// TIA Portal V20 export
FUNCTION_BLOCK "CallEquipment"   // FB131, LAD
TITLE = CallEquipment
// Template of an equipment module. This block contains the logic and futher calls (e.g. sequences, control modules, diagnostics etc.) of the equipment module.
// It can be used out of the box but also adapted to your own needs.
// stored: IsIECCheckEnabled true, MemoryReserve 100, Namespace Unit1.Em2, SetENOAutomatically true
   VAR_INPUT
      ZoneOperationEnable { ExternalWritable := 'False'} : "LWONIK_typeSafetyZoneManualOperation";
      unitEnableControlInterfaces { ExternalWritable := 'False'} : "LAF_typeEnableControlInterfaces";
      commandExcute { ExternalWritable := 'False'} : Bool;
   END_VAR
   VAR_IN_OUT
      unitStatus : "LAF_typeUnitStatus";   // Current unit status o be used in this EM
      emFeedback : "LUC_typeEmFeedback";   // Feedback of the EM to the Unit
      unitAlarmDB : "LAF_typeAlarms";   // Summarized EM Alarms for the Unit
   END_VAR
   VAR
      instSequenceSemiAutoSplice { ExternalWritable := 'False'} : "Unit1.Em2.Sequence_1_SemiAutoSplice";
      instTapeUnitInitializedJob1 { ExternalWritable := 'False'} : "LAF_SelectJob";
      instAutoSplicerModuleInitializedJob2 { ExternalWritable := 'False'} : "LAF_SelectJob";
      instLeftSplicingModuleMoverInitializedJob3 { ExternalWritable := 'False'} : "LAF_SelectJob";
      instRightSplicingModuleMoverInitializedJob4 { ExternalWritable := 'False'} : "LAF_SelectJob";
      instSplicingModuleMoverAutoJob5 { ExternalWritable := 'False'} : "LAF_SelectJob";
      instVacuumAutoJob7 { ExternalWritable := 'False'} : "LAF_SelectJob";
      instCutterAutoJob8 { ExternalWritable := 'False'} : "LAF_SelectJob";
      instLeftElectrodeReMoverAutoJob9 { ExternalWritable := 'False'} : "LAF_SelectJob";
      instRightElectrodeReMoverAutoJob10 { ExternalWritable := 'False'} : "LAF_SelectJob";
      instTapeAttachReadyAutoJob11 { ExternalWritable := 'False'} : "LAF_SelectJob";
      instTapeAttachStartAutoJob12 { ExternalWritable := 'False'} : "LAF_SelectJob";
      instTapeAttachFinishAutoJob13 { ExternalWritable := 'False'} : "LAF_SelectJob";
      instLeftSplicingModuleMoverAutoJob14 { ExternalWritable := 'False'} : "LAF_SelectJob";
      instRightSplicingModuleMoverAutoJob15 { ExternalWritable := 'False'} : "LAF_SelectJob";
      instSemiAutoSpliceFullAutoJob20 { ExternalWritable := 'False'} : "LAF_SelectJob";
      instElectrodeFixRightTopFwdBwd { ExternalWritable := 'False'} : "LBC_TwoWayActuatorCn";
      instElectrodeFixRightBottomFwdBwd { ExternalWritable := 'False'} : "LBC_TwoWayActuatorCn";
      instElectrodeFixLeftTopFwdBwd { ExternalWritable := 'False'} : "LBC_TwoWayActuatorCn";
      instElectrodeFixLeftBottomFwdBwd { ExternalWritable := 'False'} : "LBC_TwoWayActuatorCn";
      instElectrodeFixLeftTopUpDown { ExternalWritable := 'False'} : "LBC_TwoWayActuatorCn";
      instElectrodeFixLeftBottomUpDown { ExternalWritable := 'False'} : "LBC_TwoWayActuatorCn";
      instUwSemiSplicerVacuumRightTopOnOff { ExternalWritable := 'False'} : "LBC_TwoWayActuatorCn";
      instUwSemiSplicerVacuumRightBottomOnOff { ExternalWritable := 'False'} : "LBC_TwoWayActuatorCn";
      instUwSemiSplicerVacuumLeftTopOnOff { ExternalWritable := 'False'} : "LBC_TwoWayActuatorCn";
      instUwSemiSplicerVacuumLeftBottomOnOff { ExternalWritable := 'False'} : "LBC_TwoWayActuatorCn";
      instElectrodeCutterFwdBwd { ExternalWritable := 'False'} : "LBC_TwoWayActuatorCn";
      instSplicingLeftModuleMoverFwdBwd { ExternalWritable := 'False'} : "LBC_TwoWayActuatorCn";
      instSplicingRightModuleMoverFwdBwd { ExternalWritable := 'False'} : "LBC_TwoWayActuatorCn";
      instElectrodeLeftHolderMoverFwdBwd { ExternalWritable := 'False'} : "LBC_TwoWayActuatorCn";
      instElectrodeRightHolderMoverFwdBwd { ExternalWritable := 'False'} : "LBC_TwoWayActuatorCn";
      instTapeLoadingTurnCwCcw { ExternalWritable := 'False'} : "LBC_TwoWayActuatorCn";
      instTapeAttachUnitFwdBwd { ExternalWritable := 'False'} : "LBC_TwoWayActuatorCn";
      instTapeVacuumOnOff { ExternalWritable := 'False'} : "LBC_TwoWayActuatorCn";
      instStopperFwdBwd { ExternalWritable := 'False'} : "LBC_TwoWayActuatorCn";
      instSupportUnitTransferFwdBwd { ExternalWritable := 'False'} : "LBC_TwoWayActuatorCn";
      instSupportUnitShaftUpDown { ExternalWritable := 'False'} : "LBC_TwoWayActuatorCn";
      instFrameCoverFwdBwd { ExternalWritable := 'False'} : "LBC_TwoWayActuatorCn";
      statUnitStatus { ExternalWritable := 'False'} : "LAF_typeUnitStatus";   // Unit Status used in this EM
      instManageAlarms { ExternalWritable := 'False'} : "LAF_ManageAlarms";
      instEventsPFE { S7_SetPoint := 'True'} : "Unit1.Em2.EventsPFE";
      JobSummary { ExternalWritable := 'False'} : "LAF_typeJobStatus";
      statEnableManualCmds { ExternalWritable := 'False'} : Bool;
      statPulse { ExternalWritable := 'False'} : Array[0..99] of Bool;
      statTonTimer { ExternalWritable := 'False'} : Array[0..99] of TON_TIME;
      statTofTimer { ExternalWritable := 'False'} : Array[0..99] of TOF_TIME;
      citi_Ptrig : Array[0..20] of Bool;
      citiTon : Array[0..20] of TON_TIME;
      citi : Time;
      citiTest : Array[0..20] of Bool;
   END_VAR
   VAR_TEMP
      tempScInProduction : Bool;   // Mode Production and StateComplete
      tempScNoProduction : Bool;   // Mode Manual and StateComplete
   END_VAR
   VAR CONSTANT
      TO_DO_INSERT_PRECONDITIONS_HERE : Bool := TRUE;   // Template : Add em specific conditions here
      NO_JOB : DInt;   // No job
      TRUE : Bool := TRUE;
      FALSE : Bool := FALSE;
   END_VAR
   VAR_TEMP   // added for the SCL form of the ladder/FBD networks
      _w1 : Bool;
      _w2 : Bool;
   END_VAR
BEGIN

REGION Network 1: BLOCK INFO HEADER
   // (company) / (C) Copyright (year)
   // ---------------------------------------------------------------------------------
   // Title:                             (Title of this block)
   // Comment/Function: (that is implemented in the block)
   // Library/Family:           (that the source is dedicated to)
   // Author:                        (department / person in charge / contact)
   // Target System:          (test system with FW version)
   // Engineering:              TIA Portal (SW version)
   // Restrictions:               (OB types, etc.)
   // Requirements:           (hardware, technological package, etc.)
   // ---------------------------------------------------------------------------------
   // Change log table:
   // Version          | Date             | Signature      | Expert in charge  | Changes applied ------------------------|----------------------|-------------------------|--------------------------------|-----------------------
   // 001.000.000 | yyyy-mm-dd | 0x00000000 | (name of expert) | First released version
END_REGION

REGION Network 2: DESCRIPTION
   // This is a template block provided by the Automation Framework. It can be used to create an own project.
   // The Block Info Header is prepared to put in your own data.
   // Description of the block could be added here and the docu created by Code2Docu.
END_REGION

REGION Network 3: ******************** Equipment Control ********************
END_REGION

REGION Network 4: Interlink EM to Unit
   // This block links and unlinks the EM from the unit. The command to link/unlink can be set directly by the inputs of the block (e.g. to link/unlink based on any program logic) or through the InOut "hmiInterface". The block changes the output "isLinked" to true/false, depending on the command and if a change is allowed. A changed is allowed if the unit is in state aborted, clearing or stopped. The output "isLinked" is send back to the unit. If the EM is not linked, the unit ignores this EM.
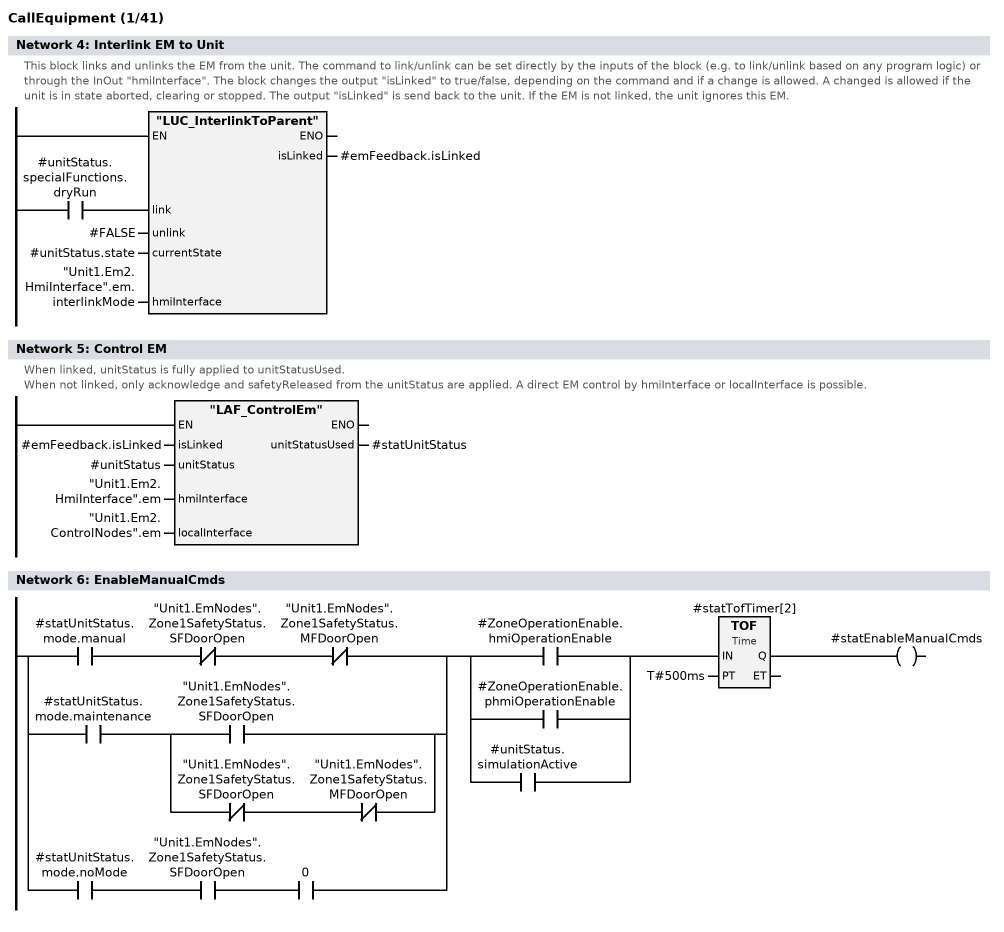
   RUNG wire#powerrail
      "LUC_InterlinkToParent"(link := wire#w1, unlink := #FALSE, currentState := #unitStatus.state, hmiInterface := "Unit1.Em2.HmiInterface".em.interlinkMode, isLinked => #emFeedback.isLinked)
   END_RUNG
   RUNG wire#powerrail
      Contact( #unitStatus.specialFunctions.dryRun )
   END_RUNG wire#w1
   // the same network as SCL:
   "LUC_InterlinkToParent"(link := #unitStatus.specialFunctions.dryRun,
                           unlink := #FALSE,
                           currentState := #unitStatus.state,
                           hmiInterface := "Unit1.Em2.HmiInterface".em.interlinkMode,
                           isLinked => #emFeedback.isLinked);
END_REGION

REGION Network 5: Control EM
   // When linked, unitStatus is fully applied to unitStatusUsed.
   // When not linked, only acknowledge and safetyReleased from the unitStatus are applied. A direct EM control by hmiInterface or localInterface is possible.
   RUNG wire#powerrail
      "LAF_ControlEm"(isLinked := #emFeedback.isLinked, unitStatus := #unitStatus, hmiInterface := "Unit1.Em2.HmiInterface".em, localInterface := "Unit1.Em2.ControlNodes".em, unitStatusUsed => #statUnitStatus)
   END_RUNG
   // the same network as SCL:
   "LAF_ControlEm"(isLinked := #emFeedback.isLinked,
                   unitStatus := #unitStatus,
                   hmiInterface := "Unit1.Em2.HmiInterface".em,
                   localInterface := "Unit1.Em2.ControlNodes".em,
                   unitStatusUsed => #statUnitStatus);
END_REGION

REGION Network 6: EnableManualCmds
   RUNG wire#powerrail
      Contact( #statUnitStatus.mode.manual )
      I_Contact( "Unit1.EmNodes".Zone1SafetyStatus.SFDoorOpen )
      I_Contact( "Unit1.EmNodes".Zone1SafetyStatus.MFDoorOpen )
      wire#w1
      Contact( #ZoneOperationEnable.hmiOperationEnable )
      wire#w3
      { S7_Templates := "time_type := Time" } #statTofTimer[2].TOF(pt := T#500ms, et =>)
      Coil( #statEnableManualCmds )
   END_RUNG
   RUNG wire#powerrail
      Contact( #statUnitStatus.mode.maintenance )
      wire#w2
      Contact( "Unit1.EmNodes".Zone1SafetyStatus.SFDoorOpen )
   END_RUNG wire#w1
   RUNG wire#w2
      I_Contact( "Unit1.EmNodes".Zone1SafetyStatus.SFDoorOpen )
      I_Contact( "Unit1.EmNodes".Zone1SafetyStatus.MFDoorOpen )
   END_RUNG wire#w1
   RUNG wire#powerrail
      Contact( #statUnitStatus.mode.noMode )
      Contact( "Unit1.EmNodes".Zone1SafetyStatus.SFDoorOpen )
      Contact( 0 )
   END_RUNG wire#w1
   RUNG wire#w1
      Contact( #ZoneOperationEnable.phmiOperationEnable )
   END_RUNG wire#w3
   RUNG wire#w1
      Contact( #unitStatus.simulationActive )
   END_RUNG wire#w3
   // the same network as SCL:
   #statTofTimer[2].TOF(IN := ((#statUnitStatus.mode.manual AND NOT "Unit1.EmNodes".Zone1SafetyStatus.SFDoorOpen AND NOT "Unit1.EmNodes".Zone1SafetyStatus.MFDoorOpen) OR (#statUnitStatus.mode.maintenance AND ("Unit1.EmNodes".Zone1SafetyStatus.SFDoorOpen OR (NOT "Unit1.EmNodes".Zone1SafetyStatus.SFDoorOpen AND NOT "Unit1.EmNodes".Zone1SafetyStatus.MFDoorOpen))) OR (#statUnitStatus.mode.noMode AND "Unit1.EmNodes".Zone1SafetyStatus.SFDoorOpen AND 0)) AND (#ZoneOperationEnable.hmiOperationEnable OR #ZoneOperationEnable.phmiOperationEnable OR #unitStatus.simulationActive),
                        PT := T#500ms);
   #statEnableManualCmds := #statTofTimer[2].Q;
END_REGION

REGION Network 7: Alarms Disabled
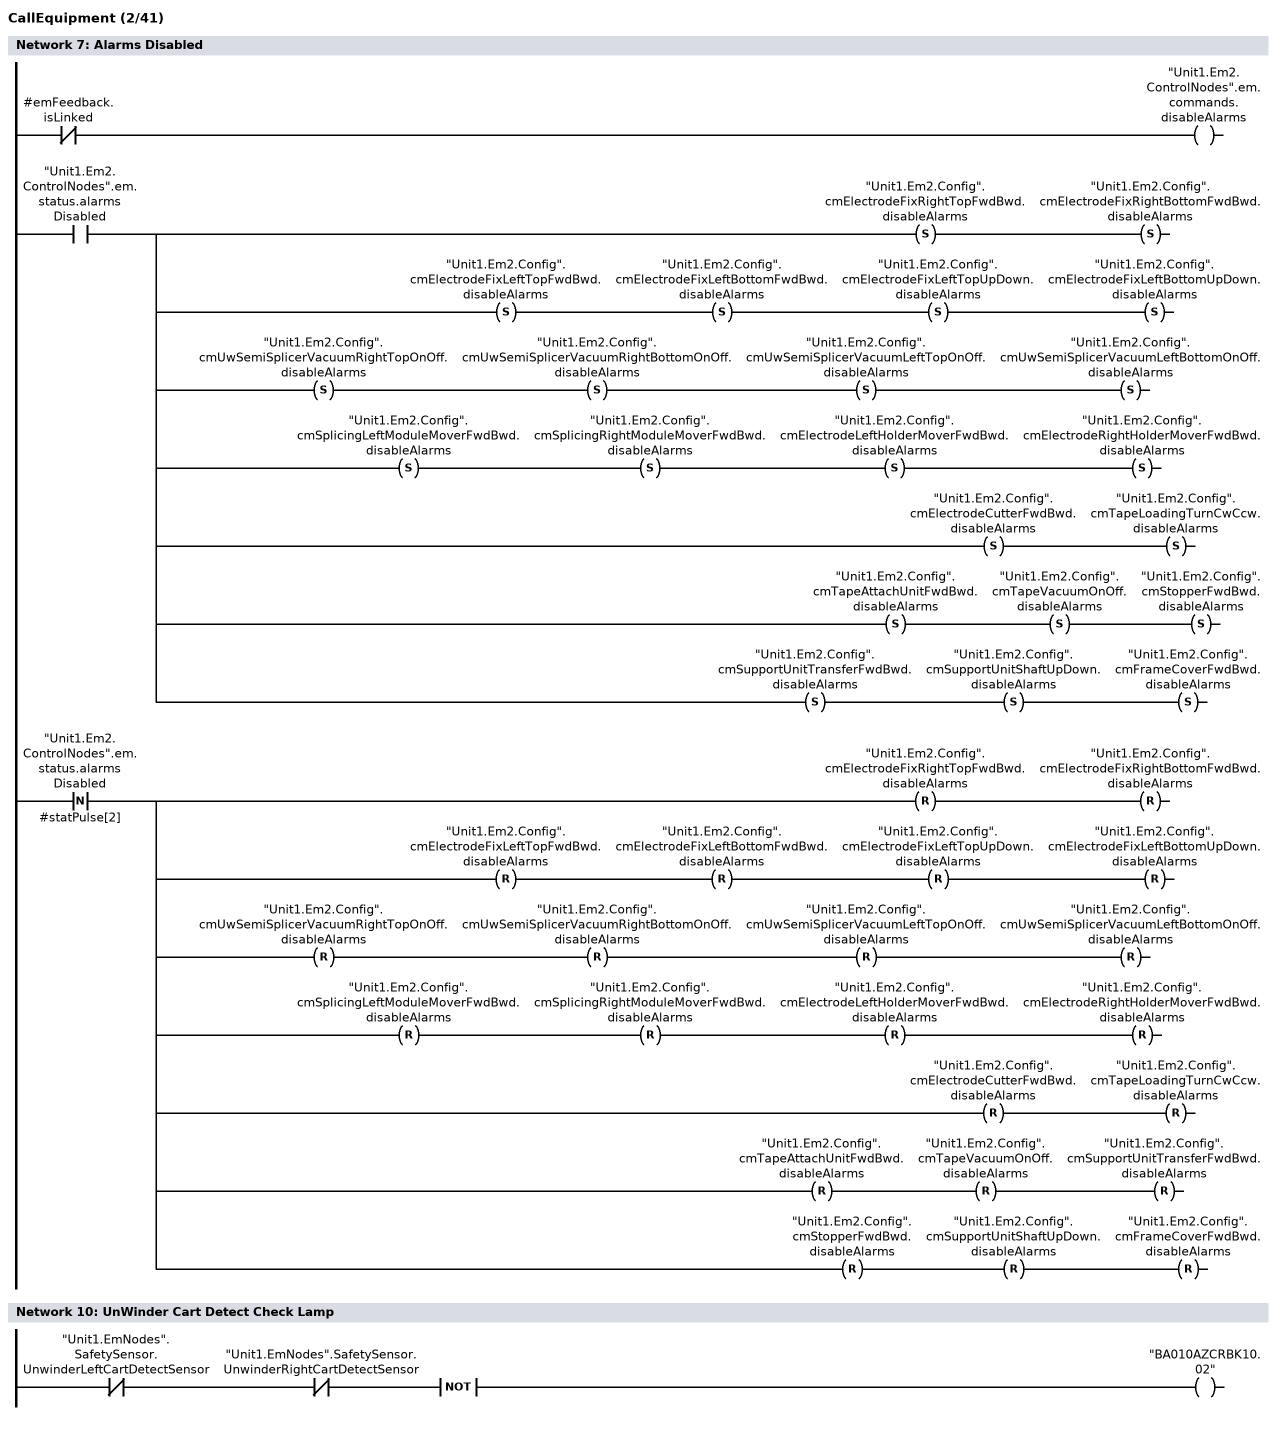
   RUNG wire#powerrail
      I_Contact( #emFeedback.isLinked )
      Coil( "Unit1.Em2.ControlNodes".em.commands.disableAlarms )
   END_RUNG
   RUNG wire#powerrail
      Contact( "Unit1.Em2.ControlNodes".em.status.alarmsDisabled )
      wire#w1
      S_Coil( "Unit1.Em2.Config".cmElectrodeFixRightTopFwdBwd.disableAlarms )
      S_Coil( "Unit1.Em2.Config".cmElectrodeFixRightBottomFwdBwd.disableAlarms )
   END_RUNG
   RUNG wire#w1
      S_Coil( "Unit1.Em2.Config".cmElectrodeFixLeftTopFwdBwd.disableAlarms )
      S_Coil( "Unit1.Em2.Config".cmElectrodeFixLeftBottomFwdBwd.disableAlarms )
      S_Coil( "Unit1.Em2.Config".cmElectrodeFixLeftTopUpDown.disableAlarms )
      S_Coil( "Unit1.Em2.Config".cmElectrodeFixLeftBottomUpDown.disableAlarms )
   END_RUNG
   RUNG wire#w1
      S_Coil( "Unit1.Em2.Config".cmUwSemiSplicerVacuumRightTopOnOff.disableAlarms )
      S_Coil( "Unit1.Em2.Config".cmUwSemiSplicerVacuumRightBottomOnOff.disableAlarms )
      S_Coil( "Unit1.Em2.Config".cmUwSemiSplicerVacuumLeftTopOnOff.disableAlarms )
      S_Coil( "Unit1.Em2.Config".cmUwSemiSplicerVacuumLeftBottomOnOff.disableAlarms )
   END_RUNG
   RUNG wire#w1
      S_Coil( "Unit1.Em2.Config".cmSplicingLeftModuleMoverFwdBwd.disableAlarms )
      S_Coil( "Unit1.Em2.Config".cmSplicingRightModuleMoverFwdBwd.disableAlarms )
      S_Coil( "Unit1.Em2.Config".cmElectrodeLeftHolderMoverFwdBwd.disableAlarms )
      S_Coil( "Unit1.Em2.Config".cmElectrodeRightHolderMoverFwdBwd.disableAlarms )
   END_RUNG
   RUNG wire#w1
      S_Coil( "Unit1.Em2.Config".cmElectrodeCutterFwdBwd.disableAlarms )
      S_Coil( "Unit1.Em2.Config".cmTapeLoadingTurnCwCcw.disableAlarms )
   END_RUNG
   RUNG wire#w1
      S_Coil( "Unit1.Em2.Config".cmTapeAttachUnitFwdBwd.disableAlarms )
      S_Coil( "Unit1.Em2.Config".cmTapeVacuumOnOff.disableAlarms )
      S_Coil( "Unit1.Em2.Config".cmStopperFwdBwd.disableAlarms )
   END_RUNG
   RUNG wire#w1
      S_Coil( "Unit1.Em2.Config".cmSupportUnitTransferFwdBwd.disableAlarms )
      S_Coil( "Unit1.Em2.Config".cmSupportUnitShaftUpDown.disableAlarms )
      S_Coil( "Unit1.Em2.Config".cmFrameCoverFwdBwd.disableAlarms )
   END_RUNG
   RUNG wire#powerrail
      N_Contact(operand := "Unit1.Em2.ControlNodes".em.status.alarmsDisabled, bit := #statPulse[2])
      wire#w2
      R_Coil( "Unit1.Em2.Config".cmElectrodeFixRightTopFwdBwd.disableAlarms )
      R_Coil( "Unit1.Em2.Config".cmElectrodeFixRightBottomFwdBwd.disableAlarms )
   END_RUNG
   RUNG wire#w2
      R_Coil( "Unit1.Em2.Config".cmElectrodeFixLeftTopFwdBwd.disableAlarms )
      R_Coil( "Unit1.Em2.Config".cmElectrodeFixLeftBottomFwdBwd.disableAlarms )
      R_Coil( "Unit1.Em2.Config".cmElectrodeFixLeftTopUpDown.disableAlarms )
      R_Coil( "Unit1.Em2.Config".cmElectrodeFixLeftBottomUpDown.disableAlarms )
   END_RUNG
   RUNG wire#w2
      R_Coil( "Unit1.Em2.Config".cmUwSemiSplicerVacuumRightTopOnOff.disableAlarms )
      R_Coil( "Unit1.Em2.Config".cmUwSemiSplicerVacuumRightBottomOnOff.disableAlarms )
      R_Coil( "Unit1.Em2.Config".cmUwSemiSplicerVacuumLeftTopOnOff.disableAlarms )
      R_Coil( "Unit1.Em2.Config".cmUwSemiSplicerVacuumLeftBottomOnOff.disableAlarms )
   END_RUNG
   RUNG wire#w2
      R_Coil( "Unit1.Em2.Config".cmSplicingLeftModuleMoverFwdBwd.disableAlarms )
      R_Coil( "Unit1.Em2.Config".cmSplicingRightModuleMoverFwdBwd.disableAlarms )
      R_Coil( "Unit1.Em2.Config".cmElectrodeLeftHolderMoverFwdBwd.disableAlarms )
      R_Coil( "Unit1.Em2.Config".cmElectrodeRightHolderMoverFwdBwd.disableAlarms )
   END_RUNG
   RUNG wire#w2
      R_Coil( "Unit1.Em2.Config".cmElectrodeCutterFwdBwd.disableAlarms )
      R_Coil( "Unit1.Em2.Config".cmTapeLoadingTurnCwCcw.disableAlarms )
   END_RUNG
   RUNG wire#w2
      R_Coil( "Unit1.Em2.Config".cmTapeAttachUnitFwdBwd.disableAlarms )
      R_Coil( "Unit1.Em2.Config".cmTapeVacuumOnOff.disableAlarms )
      R_Coil( "Unit1.Em2.Config".cmSupportUnitTransferFwdBwd.disableAlarms )
   END_RUNG
   RUNG wire#w2
      R_Coil( "Unit1.Em2.Config".cmStopperFwdBwd.disableAlarms )
      R_Coil( "Unit1.Em2.Config".cmSupportUnitShaftUpDown.disableAlarms )
      R_Coil( "Unit1.Em2.Config".cmFrameCoverFwdBwd.disableAlarms )
   END_RUNG
   // the same network as SCL:
   "Unit1.Em2.ControlNodes".em.commands.disableAlarms := NOT #emFeedback.isLinked;
   IF "Unit1.Em2.ControlNodes".em.status.alarmsDisabled THEN
       "Unit1.Em2.Config".cmElectrodeFixRightTopFwdBwd.disableAlarms := TRUE;
       "Unit1.Em2.Config".cmElectrodeFixRightBottomFwdBwd.disableAlarms := TRUE;
       "Unit1.Em2.Config".cmElectrodeFixLeftTopFwdBwd.disableAlarms := TRUE;
       "Unit1.Em2.Config".cmElectrodeFixLeftBottomFwdBwd.disableAlarms := TRUE;
       "Unit1.Em2.Config".cmElectrodeFixLeftTopUpDown.disableAlarms := TRUE;
       "Unit1.Em2.Config".cmElectrodeFixLeftBottomUpDown.disableAlarms := TRUE;
       "Unit1.Em2.Config".cmUwSemiSplicerVacuumRightTopOnOff.disableAlarms := TRUE;
       "Unit1.Em2.Config".cmUwSemiSplicerVacuumRightBottomOnOff.disableAlarms := TRUE;
       "Unit1.Em2.Config".cmUwSemiSplicerVacuumLeftTopOnOff.disableAlarms := TRUE;
       "Unit1.Em2.Config".cmUwSemiSplicerVacuumLeftBottomOnOff.disableAlarms := TRUE;
       "Unit1.Em2.Config".cmSplicingLeftModuleMoverFwdBwd.disableAlarms := TRUE;
       "Unit1.Em2.Config".cmSplicingRightModuleMoverFwdBwd.disableAlarms := TRUE;
       "Unit1.Em2.Config".cmElectrodeLeftHolderMoverFwdBwd.disableAlarms := TRUE;
       "Unit1.Em2.Config".cmElectrodeRightHolderMoverFwdBwd.disableAlarms := TRUE;
       "Unit1.Em2.Config".cmElectrodeCutterFwdBwd.disableAlarms := TRUE;
       "Unit1.Em2.Config".cmTapeLoadingTurnCwCcw.disableAlarms := TRUE;
       "Unit1.Em2.Config".cmTapeAttachUnitFwdBwd.disableAlarms := TRUE;
       "Unit1.Em2.Config".cmTapeVacuumOnOff.disableAlarms := TRUE;
       "Unit1.Em2.Config".cmStopperFwdBwd.disableAlarms := TRUE;
       "Unit1.Em2.Config".cmSupportUnitTransferFwdBwd.disableAlarms := TRUE;
       "Unit1.Em2.Config".cmSupportUnitShaftUpDown.disableAlarms := TRUE;
       "Unit1.Em2.Config".cmFrameCoverFwdBwd.disableAlarms := TRUE;
   END_IF;
   #_w1 := NOT "Unit1.Em2.ControlNodes".em.status.alarmsDisabled AND #statPulse[2];   // falling edge of "Unit1.Em2.ControlNodes".em.status.alarmsDisabled
   #statPulse[2] := "Unit1.Em2.ControlNodes".em.status.alarmsDisabled;
   IF #_w1 THEN
       "Unit1.Em2.Config".cmElectrodeFixRightTopFwdBwd.disableAlarms := FALSE;
       "Unit1.Em2.Config".cmElectrodeFixRightBottomFwdBwd.disableAlarms := FALSE;
       "Unit1.Em2.Config".cmElectrodeFixLeftTopFwdBwd.disableAlarms := FALSE;
       "Unit1.Em2.Config".cmElectrodeFixLeftBottomFwdBwd.disableAlarms := FALSE;
       "Unit1.Em2.Config".cmElectrodeFixLeftTopUpDown.disableAlarms := FALSE;
       "Unit1.Em2.Config".cmElectrodeFixLeftBottomUpDown.disableAlarms := FALSE;
       "Unit1.Em2.Config".cmUwSemiSplicerVacuumRightTopOnOff.disableAlarms := FALSE;
       "Unit1.Em2.Config".cmUwSemiSplicerVacuumRightBottomOnOff.disableAlarms := FALSE;
       "Unit1.Em2.Config".cmUwSemiSplicerVacuumLeftTopOnOff.disableAlarms := FALSE;
       "Unit1.Em2.Config".cmUwSemiSplicerVacuumLeftBottomOnOff.disableAlarms := FALSE;
       "Unit1.Em2.Config".cmSplicingLeftModuleMoverFwdBwd.disableAlarms := FALSE;
       "Unit1.Em2.Config".cmSplicingRightModuleMoverFwdBwd.disableAlarms := FALSE;
       "Unit1.Em2.Config".cmElectrodeLeftHolderMoverFwdBwd.disableAlarms := FALSE;
       "Unit1.Em2.Config".cmElectrodeRightHolderMoverFwdBwd.disableAlarms := FALSE;
       "Unit1.Em2.Config".cmElectrodeCutterFwdBwd.disableAlarms := FALSE;
       "Unit1.Em2.Config".cmTapeLoadingTurnCwCcw.disableAlarms := FALSE;
       "Unit1.Em2.Config".cmTapeAttachUnitFwdBwd.disableAlarms := FALSE;
       "Unit1.Em2.Config".cmTapeVacuumOnOff.disableAlarms := FALSE;
       "Unit1.Em2.Config".cmSupportUnitTransferFwdBwd.disableAlarms := FALSE;
       "Unit1.Em2.Config".cmStopperFwdBwd.disableAlarms := FALSE;
       "Unit1.Em2.Config".cmSupportUnitShaftUpDown.disableAlarms := FALSE;
       "Unit1.Em2.Config".cmFrameCoverFwdBwd.disableAlarms := FALSE;
   END_IF;
END_REGION

REGION Network 8 (SCL): ReferenceDesignator
   IF "Unit1.EmNodes".unitRecipe.processUnitNo = 2 THEN
       "Unit1.Em2.Config".cmElectrodeFixRightTopFwdBwd.referenceDesignator := WSTRING#'Electrode Fix Right Top';
       "Unit1.Em2.Config".cmElectrodeFixRightBottomFwdBwd.referenceDesignator := WSTRING#'Electrode Fix Right BTM';
       "Unit1.Em2.Config".cmElectrodeFixLeftTopFwdBwd.referenceDesignator := WSTRING#'Electrode Fix Left Top';
       "Unit1.Em2.Config".cmElectrodeFixLeftBottomFwdBwd.referenceDesignator := WSTRING#'Electrode Fix Left BTM';
       "Unit1.Em2.Config".cmElectrodeFixLeftTopUpDown.referenceDesignator := WSTRING#'Electrode Fix Left Top';
       "Unit1.Em2.Config".cmElectrodeFixLeftBottomUpDown.referenceDesignator := WSTRING#'Electrode Fix Left BTM';
       "Unit1.Em2.Config".cmUwSemiSplicerVacuumRightTopOnOff.referenceDesignator := WSTRING#'Splicer Vacuum Right Top';
       "Unit1.Em2.Config".cmUwSemiSplicerVacuumRightBottomOnOff.referenceDesignator := WSTRING#'Splicer Vacuum Right BTM';
       "Unit1.Em2.Config".cmUwSemiSplicerVacuumLeftTopOnOff.referenceDesignator := WSTRING#'Splicer Vacuum Left Top';
       "Unit1.Em2.Config".cmUwSemiSplicerVacuumLeftBottomOnOff.referenceDesignator := WSTRING#'Splicer Vacuum Left BTM';
       "Unit1.Em2.Config".cmElectrodeCutterFwdBwd.referenceDesignator := WSTRING#'Electrode Cutter';
       "Unit1.Em2.Config".cmSplicingLeftModuleMoverFwdBwd.referenceDesignator := WSTRING#'Left Module Mover';
       "Unit1.Em2.Config".cmSplicingRightModuleMoverFwdBwd.referenceDesignator := WSTRING#'Right Module Mover';
       "Unit1.Em2.Config".cmElectrodeLeftHolderMoverFwdBwd.referenceDesignator := WSTRING#'Left Holder Mover';
       "Unit1.Em2.Config".cmElectrodeRightHolderMoverFwdBwd.referenceDesignator := WSTRING#'Right Holder Mover';
       "Unit1.Em2.Config".cmTapeLoadingTurnCwCcw.referenceDesignator := WSTRING#'Tape Loading Tum';
       "Unit1.Em2.Config".cmTapeAttachUnitFwdBwd.referenceDesignator := WSTRING#'Tape Attach Unit';
       "Unit1.Em2.Config".cmTapeVacuumOnOff.referenceDesignator := WSTRING#'Tape Vacuum';
       "Unit1.Em2.Config".cmStopperFwdBwd.referenceDesignator := WSTRING#'Stopper';
       "Unit1.Em2.Config".cmSupportUnitTransferFwdBwd.referenceDesignator := WSTRING#'Support Unit Transfer';
       "Unit1.Em2.Config".cmSupportUnitShaftUpDown.referenceDesignator := WSTRING#'Support Unit Shaft';
       "Unit1.Em2.Config".cmFrameCoverFwdBwd.referenceDesignator := WSTRING#'Frame Cover';
   END_IF;

   IF "Unit1.EmNodes".unitRecipe.processUnitNo = 1 THEN
       "Unit1.Em2.Config".cmElectrodeFixRightTopFwdBwd.referenceDesignator := WSTRING#'Electrode Fix Left Top';
       "Unit1.Em2.Config".cmElectrodeFixRightBottomFwdBwd.referenceDesignator := WSTRING#'Electrode Fix Left BTM';
       "Unit1.Em2.Config".cmElectrodeFixLeftTopFwdBwd.referenceDesignator := WSTRING#'Electrode Fix Right Top';
       "Unit1.Em2.Config".cmElectrodeFixLeftBottomFwdBwd.referenceDesignator := WSTRING#'Electrode Fix Right BTM';
       "Unit1.Em2.Config".cmElectrodeFixLeftTopUpDown.referenceDesignator := WSTRING#'Electrode Fix Right Top';
       "Unit1.Em2.Config".cmElectrodeFixLeftBottomUpDown.referenceDesignator := WSTRING#'Electrode Fix Right BTM';
       "Unit1.Em2.Config".cmUwSemiSplicerVacuumRightTopOnOff.referenceDesignator := WSTRING#'Splicer Vacuum Left Top';
       "Unit1.Em2.Config".cmUwSemiSplicerVacuumRightBottomOnOff.referenceDesignator := WSTRING#'Splicer Vacuum Left BTM';
       "Unit1.Em2.Config".cmUwSemiSplicerVacuumLeftTopOnOff.referenceDesignator := WSTRING#'Splicer Vacuum Right Top';
       "Unit1.Em2.Config".cmUwSemiSplicerVacuumLeftBottomOnOff.referenceDesignator := WSTRING#'Splicer Vacuum Right BTM';
       "Unit1.Em2.Config".cmElectrodeCutterFwdBwd.referenceDesignator := WSTRING#'Electrode Cutter';
       "Unit1.Em2.Config".cmSplicingLeftModuleMoverFwdBwd.referenceDesignator := WSTRING#'Right Module Mover';
       "Unit1.Em2.Config".cmSplicingRightModuleMoverFwdBwd.referenceDesignator := WSTRING#'Left Module Mover';
       "Unit1.Em2.Config".cmElectrodeLeftHolderMoverFwdBwd.referenceDesignator := WSTRING#'Right Holder Mover';
       "Unit1.Em2.Config".cmElectrodeRightHolderMoverFwdBwd.referenceDesignator := WSTRING#'Left Holder Mover';
       "Unit1.Em2.Config".cmTapeLoadingTurnCwCcw.referenceDesignator := WSTRING#'Tape Loading Tum';
       "Unit1.Em2.Config".cmTapeAttachUnitFwdBwd.referenceDesignator := WSTRING#'Tape Attach Unit';
       "Unit1.Em2.Config".cmTapeVacuumOnOff.referenceDesignator := WSTRING#'Tape Vacuum';
       "Unit1.Em2.Config".cmStopperFwdBwd.referenceDesignator := WSTRING#'Stopper';
       "Unit1.Em2.Config".cmSupportUnitTransferFwdBwd.referenceDesignator := WSTRING#'Support Unit Transfer';
       "Unit1.Em2.Config".cmSupportUnitShaftUpDown.referenceDesignator := WSTRING#'Support Unit Shaft';
       "Unit1.Em2.Config".cmFrameCoverFwdBwd.referenceDesignator := WSTRING#'Frame Cover';
   END_IF;
END_REGION

REGION Network 9: ******************** Control Modules (Sensors) ********************
   // Call control modules that are sensors before the em logic (jobs and sequence), so that the latest value is used in the logic.
END_REGION

REGION Network 10: UnWinder Cart Detect Check Lamp
   RUNG wire#powerrail
      I_Contact( "Unit1.EmNodes".SafetySensor.UnwinderLeftCartDetectSensor )
      I_Contact( "Unit1.EmNodes".SafetySensor.UnwinderRightCartDetectSensor )
      Not()
      Coil( "BA010AZCRBK10.02" )
   END_RUNG
   // the same network as SCL:
   "BA010AZCRBK10.02" := NOT (NOT "Unit1.EmNodes".SafetySensor.UnwinderLeftCartDetectSensor AND NOT "Unit1.EmNodes".SafetySensor.UnwinderRightCartDetectSensor);
END_REGION

REGION Network 11: ******************** Equipment Logic ********************
   // Title:
   // Comment/Function:
   // Author:
   // Engineering:
   // Restrictions:
   // Requirements:
END_REGION

REGION Network 12: Map Unit Status to Sequence Status [1] Semi Auto Splice
   // This block maps the unit status to the seuqnce status. Thus, it controls the sequence depending on the unit status. E.g. it sets the sequence to automatic when the unit state is in productions. This blocks work perfectly with the sequences provided in the AF. 
   // This typed block (MapUnitStatusToSequence) could be adjusted to specific application requirements or if other, user-defined sequences are used.
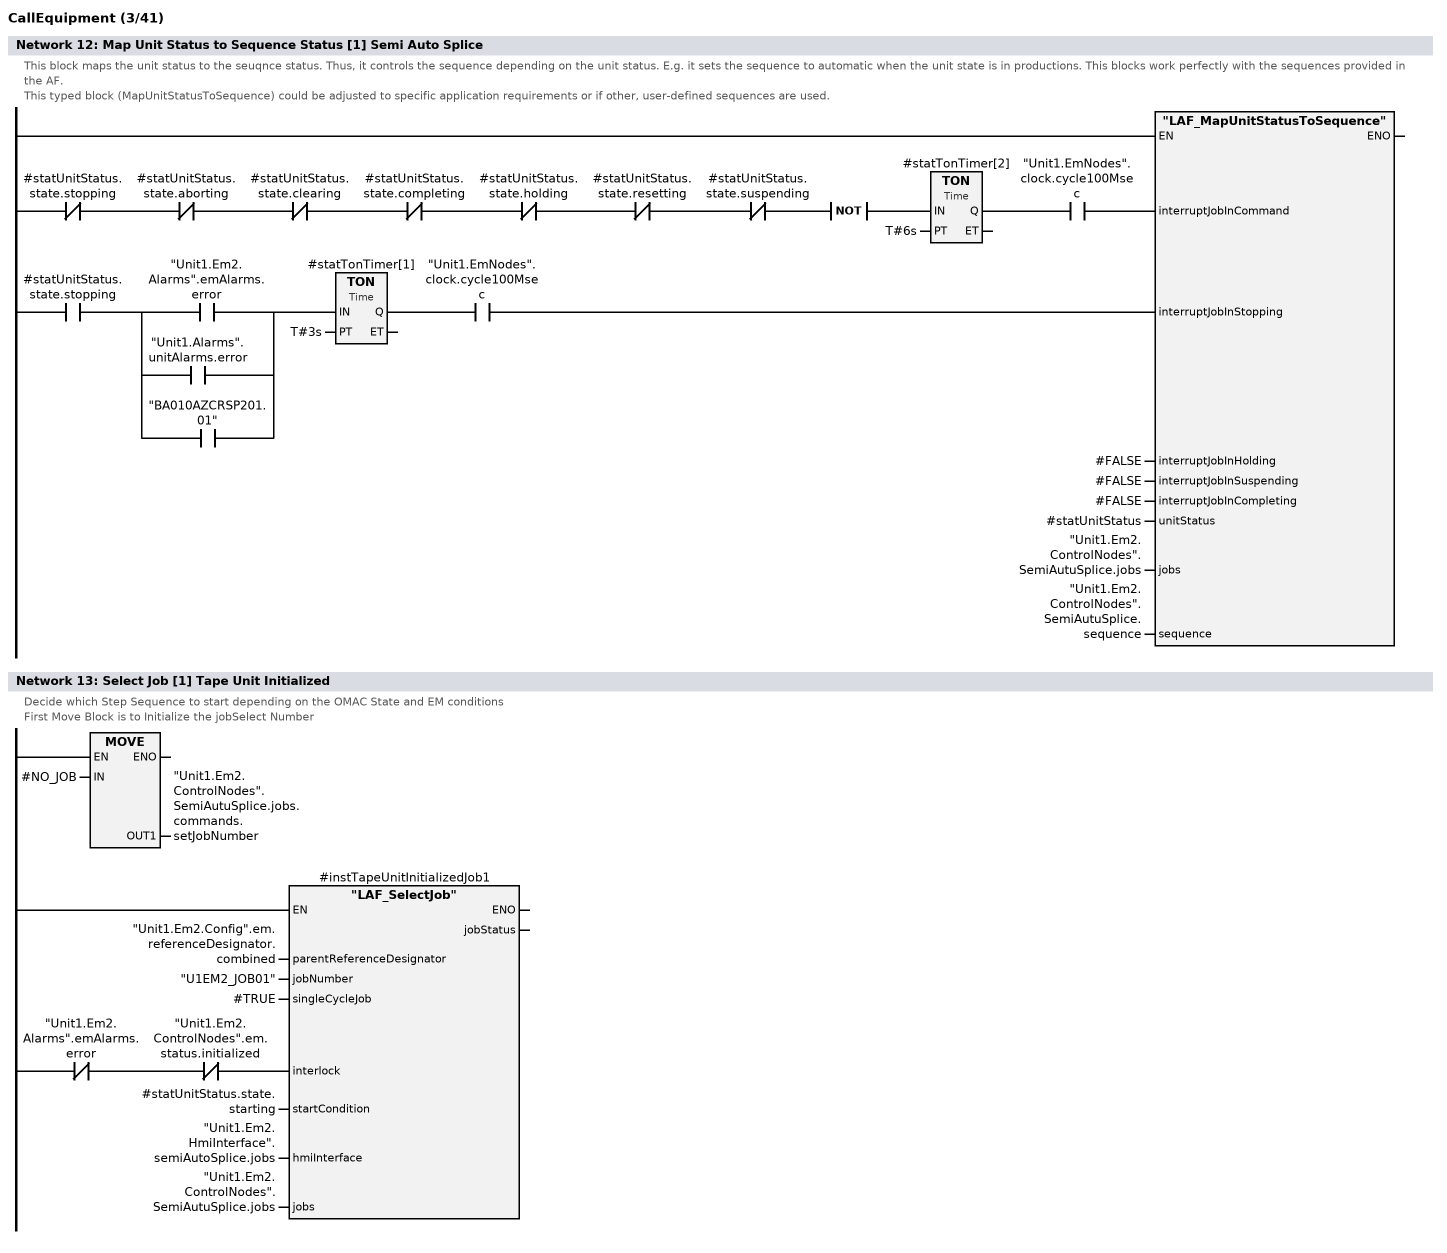
   RUNG wire#powerrail
      "LAF_MapUnitStatusToSequence"(interruptJobInCommand := wire#w1, interruptJobInStopping := wire#w4, interruptJobInHolding := #FALSE, interruptJobInSuspending := #FALSE, interruptJobInCompleting := #FALSE, unitStatus := #statUnitStatus, jobs := "Unit1.Em2.ControlNodes".SemiAutuSplice.jobs, sequence := "Unit1.Em2.ControlNodes".SemiAutuSplice.sequence)
   END_RUNG
   RUNG wire#powerrail
      I_Contact( #statUnitStatus.state.stopping )
      I_Contact( #statUnitStatus.state.aborting )
      I_Contact( #statUnitStatus.state.clearing )
      I_Contact( #statUnitStatus.state.completing )
      I_Contact( #statUnitStatus.state.holding )
      I_Contact( #statUnitStatus.state.resetting )
      I_Contact( #statUnitStatus.state.suspending )
      Not()
      { S7_Templates := "time_type := Time" } #statTonTimer[2].TON(pt := T#6s, et =>)
      Contact( "Unit1.EmNodes".clock.cycle100Msec )
   END_RUNG wire#w1
   RUNG wire#powerrail
      Contact( #statUnitStatus.state.stopping )
      wire#w2
      Contact( "Unit1.Em2.Alarms".emAlarms.error )
      wire#w3
      { S7_Templates := "time_type := Time" } #statTonTimer[1].TON(pt := T#3s, et =>)
      Contact( "Unit1.EmNodes".clock.cycle100Msec )
   END_RUNG wire#w4
   RUNG wire#w2
      Contact( "Unit1.Alarms".unitAlarms.error )
   END_RUNG wire#w3
   RUNG wire#w2
      Contact( "BA010AZCRSP201.01" )
   END_RUNG wire#w3
   // the same network as SCL:
   #statTonTimer[2].TON(IN := NOT (NOT #statUnitStatus.state.stopping AND NOT #statUnitStatus.state.aborting AND NOT #statUnitStatus.state.clearing AND NOT #statUnitStatus.state.completing AND NOT #statUnitStatus.state.holding AND NOT #statUnitStatus.state.resetting AND NOT #statUnitStatus.state.suspending),
                        PT := T#6s);
   #_w1 := #statTonTimer[2].Q AND "Unit1.EmNodes".clock.cycle100Msec;
   #statTonTimer[1].TON(IN := #statUnitStatus.state.stopping AND ("Unit1.Em2.Alarms".emAlarms.error OR "Unit1.Alarms".unitAlarms.error OR "BA010AZCRSP201.01"),
                        PT := T#3s);
   "LAF_MapUnitStatusToSequence"(interruptJobInCommand := #_w1,
                           interruptJobInStopping := #statTonTimer[1].Q AND "Unit1.EmNodes".clock.cycle100Msec,
                           interruptJobInHolding := #FALSE,
                           interruptJobInSuspending := #FALSE,
                           interruptJobInCompleting := #FALSE,
                           unitStatus := #statUnitStatus,
                           jobs := "Unit1.Em2.ControlNodes".SemiAutuSplice.jobs,
                           sequence := "Unit1.Em2.ControlNodes".SemiAutuSplice.sequence);
END_REGION

REGION Network 13: Select Job [1] Tape Unit Initialized
   // Decide which Step Sequence to start depending on the OMAC State and EM conditions
   // First Move Block is to Initialize the jobSelect Number
   RUNG wire#powerrail
      Move(in := #NO_JOB, out1 => "Unit1.Em2.ControlNodes".SemiAutuSplice.jobs.commands.setJobNumber)
   END_RUNG
   RUNG wire#powerrail
      #instTapeUnitInitializedJob1(interlock := wire#w1, parentReferenceDesignator := "Unit1.Em2.Config".em.referenceDesignator.combined, jobNumber := "U1EM2_JOB01", singleCycleJob := #TRUE, startCondition := #statUnitStatus.state.starting, hmiInterface := "Unit1.Em2.HmiInterface".semiAutoSplice.jobs, jobs := "Unit1.Em2.ControlNodes".SemiAutuSplice.jobs, jobStatus =>)
   END_RUNG
   RUNG wire#powerrail
      I_Contact( "Unit1.Em2.Alarms".emAlarms.error )
      I_Contact( "Unit1.Em2.ControlNodes".em.status.initialized )
   END_RUNG wire#w1
   // the same network as SCL:
   "Unit1.Em2.ControlNodes".SemiAutuSplice.jobs.commands.setJobNumber := #NO_JOB;
   #instTapeUnitInitializedJob1(parentReferenceDesignator := "Unit1.Em2.Config".em.referenceDesignator.combined,   // "LAF_SelectJob"
                           jobNumber := "U1EM2_JOB01",
                           singleCycleJob := #TRUE,
                           interlock := NOT "Unit1.Em2.Alarms".emAlarms.error AND NOT "Unit1.Em2.ControlNodes".em.status.initialized,
                           startCondition := #statUnitStatus.state.starting,
                           hmiInterface := "Unit1.Em2.HmiInterface".semiAutoSplice.jobs,
                           jobs := "Unit1.Em2.ControlNodes".SemiAutuSplice.jobs);
END_REGION

REGION Network 14: Select Job [2] Auto Splicer Module Initialized
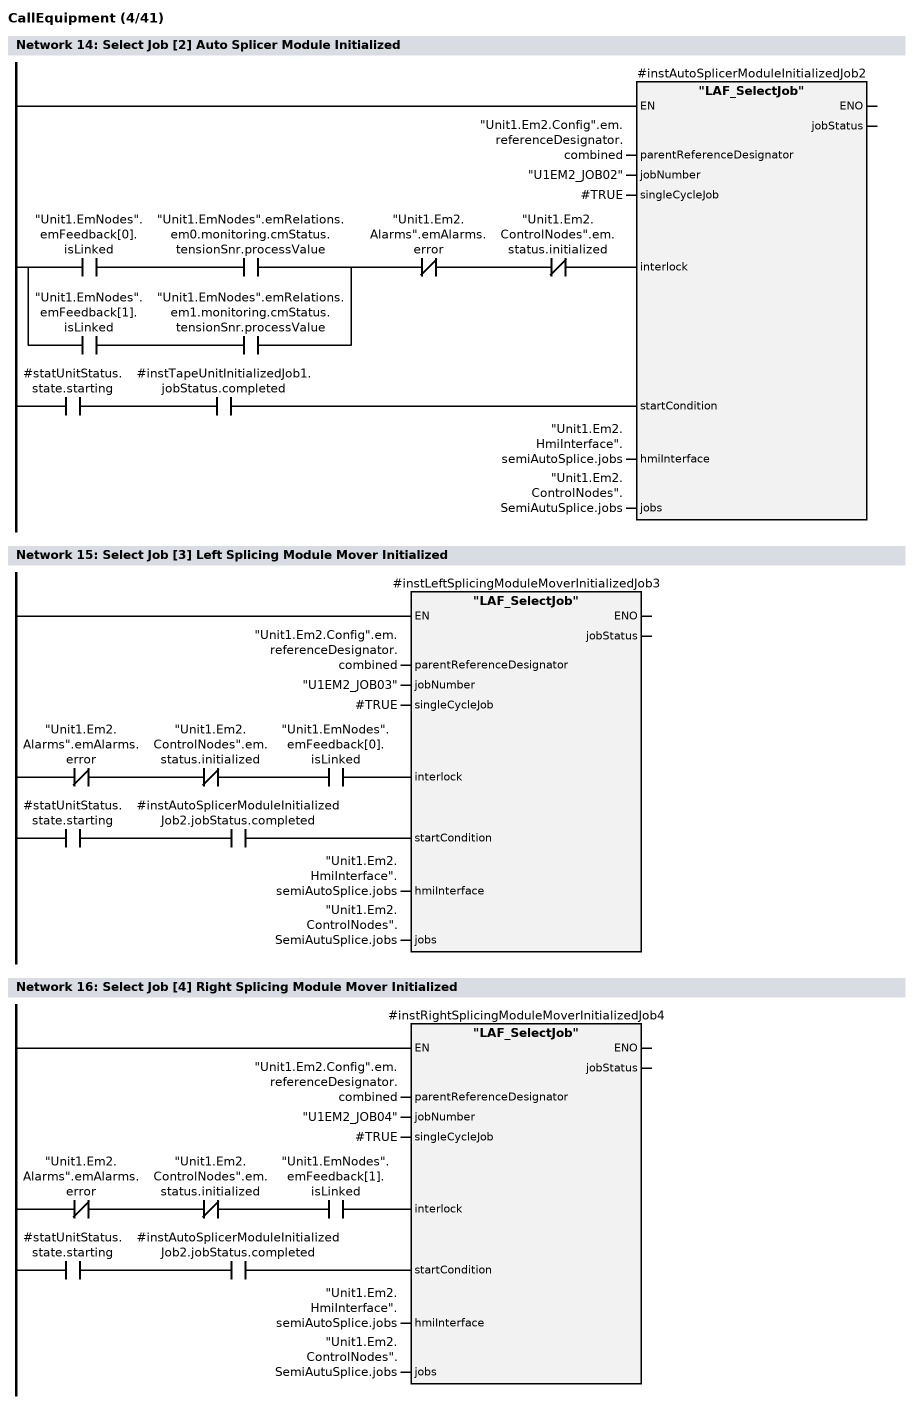
   RUNG wire#powerrail
      #instAutoSplicerModuleInitializedJob2(interlock := wire#w2, startCondition := wire#w3, parentReferenceDesignator := "Unit1.Em2.Config".em.referenceDesignator.combined, jobNumber := "U1EM2_JOB02", singleCycleJob := #TRUE, hmiInterface := "Unit1.Em2.HmiInterface".semiAutoSplice.jobs, jobs := "Unit1.Em2.ControlNodes".SemiAutuSplice.jobs, jobStatus =>)
   END_RUNG
   RUNG wire#powerrail
      Contact( "Unit1.EmNodes".emFeedback[0].isLinked )
      Contact( "Unit1.EmNodes".emRelations.em0.monitoring.cmStatus.tensionSnr.processValue )
      wire#w1
      I_Contact( "Unit1.Em2.Alarms".emAlarms.error )
      I_Contact( "Unit1.Em2.ControlNodes".em.status.initialized )
   END_RUNG wire#w2
   RUNG wire#powerrail
      Contact( "Unit1.EmNodes".emFeedback[1].isLinked )
      Contact( "Unit1.EmNodes".emRelations.em1.monitoring.cmStatus.tensionSnr.processValue )
   END_RUNG wire#w1
   RUNG wire#powerrail
      Contact( #statUnitStatus.state.starting )
      Contact( #instTapeUnitInitializedJob1.jobStatus.completed )
   END_RUNG wire#w3
   // the same network as SCL:
   #instAutoSplicerModuleInitializedJob2(parentReferenceDesignator := "Unit1.Em2.Config".em.referenceDesignator.combined,   // "LAF_SelectJob"
                           jobNumber := "U1EM2_JOB02",
                           singleCycleJob := #TRUE,
                           interlock := (("Unit1.EmNodes".emFeedback[0].isLinked AND "Unit1.EmNodes".emRelations.em0.monitoring.cmStatus.tensionSnr.processValue) OR ("Unit1.EmNodes".emFeedback[1].isLinked AND "Unit1.EmNodes".emRelations.em1.monitoring.cmStatus.tensionSnr.processValue)) AND NOT "Unit1.Em2.Alarms".emAlarms.error AND NOT "Unit1.Em2.ControlNodes".em.status.initialized,
                           startCondition := #statUnitStatus.state.starting AND #instTapeUnitInitializedJob1.jobStatus.completed,
                           hmiInterface := "Unit1.Em2.HmiInterface".semiAutoSplice.jobs,
                           jobs := "Unit1.Em2.ControlNodes".SemiAutuSplice.jobs);
END_REGION

REGION Network 15: Select Job [3] Left Splicing Module Mover Initialized
   RUNG wire#powerrail
      #instLeftSplicingModuleMoverInitializedJob3(interlock := wire#w1, startCondition := wire#w2, parentReferenceDesignator := "Unit1.Em2.Config".em.referenceDesignator.combined, jobNumber := "U1EM2_JOB03", singleCycleJob := #TRUE, hmiInterface := "Unit1.Em2.HmiInterface".semiAutoSplice.jobs, jobs := "Unit1.Em2.ControlNodes".SemiAutuSplice.jobs, jobStatus =>)
   END_RUNG
   RUNG wire#powerrail
      I_Contact( "Unit1.Em2.Alarms".emAlarms.error )
      I_Contact( "Unit1.Em2.ControlNodes".em.status.initialized )
      Contact( "Unit1.EmNodes".emFeedback[0].isLinked )
   END_RUNG wire#w1
   RUNG wire#powerrail
      Contact( #statUnitStatus.state.starting )
      Contact( #instAutoSplicerModuleInitializedJob2.jobStatus.completed )
   END_RUNG wire#w2
   // the same network as SCL:
   #instLeftSplicingModuleMoverInitializedJob3(parentReferenceDesignator := "Unit1.Em2.Config".em.referenceDesignator.combined,   // "LAF_SelectJob"
                           jobNumber := "U1EM2_JOB03",
                           singleCycleJob := #TRUE,
                           interlock := NOT "Unit1.Em2.Alarms".emAlarms.error AND NOT "Unit1.Em2.ControlNodes".em.status.initialized AND "Unit1.EmNodes".emFeedback[0].isLinked,
                           startCondition := #statUnitStatus.state.starting AND #instAutoSplicerModuleInitializedJob2.jobStatus.completed,
                           hmiInterface := "Unit1.Em2.HmiInterface".semiAutoSplice.jobs,
                           jobs := "Unit1.Em2.ControlNodes".SemiAutuSplice.jobs);
END_REGION

REGION Network 16: Select Job [4] Right Splicing Module Mover Initialized
   RUNG wire#powerrail
      #instRightSplicingModuleMoverInitializedJob4(interlock := wire#w1, startCondition := wire#w2, parentReferenceDesignator := "Unit1.Em2.Config".em.referenceDesignator.combined, jobNumber := "U1EM2_JOB04", singleCycleJob := #TRUE, hmiInterface := "Unit1.Em2.HmiInterface".semiAutoSplice.jobs, jobs := "Unit1.Em2.ControlNodes".SemiAutuSplice.jobs, jobStatus =>)
   END_RUNG
   RUNG wire#powerrail
      I_Contact( "Unit1.Em2.Alarms".emAlarms.error )
      I_Contact( "Unit1.Em2.ControlNodes".em.status.initialized )
      Contact( "Unit1.EmNodes".emFeedback[1].isLinked )
   END_RUNG wire#w1
   RUNG wire#powerrail
      Contact( #statUnitStatus.state.starting )
      Contact( #instAutoSplicerModuleInitializedJob2.jobStatus.completed )
   END_RUNG wire#w2
   // the same network as SCL:
   #instRightSplicingModuleMoverInitializedJob4(parentReferenceDesignator := "Unit1.Em2.Config".em.referenceDesignator.combined,   // "LAF_SelectJob"
                           jobNumber := "U1EM2_JOB04",
                           singleCycleJob := #TRUE,
                           interlock := NOT "Unit1.Em2.Alarms".emAlarms.error AND NOT "Unit1.Em2.ControlNodes".em.status.initialized AND "Unit1.EmNodes".emFeedback[1].isLinked,
                           startCondition := #statUnitStatus.state.starting AND #instAutoSplicerModuleInitializedJob2.jobStatus.completed,
                           hmiInterface := "Unit1.Em2.HmiInterface".semiAutoSplice.jobs,
                           jobs := "Unit1.Em2.ControlNodes".SemiAutuSplice.jobs);
END_REGION

REGION Network 17: Select Job [5] Splicing Module Mover Auto
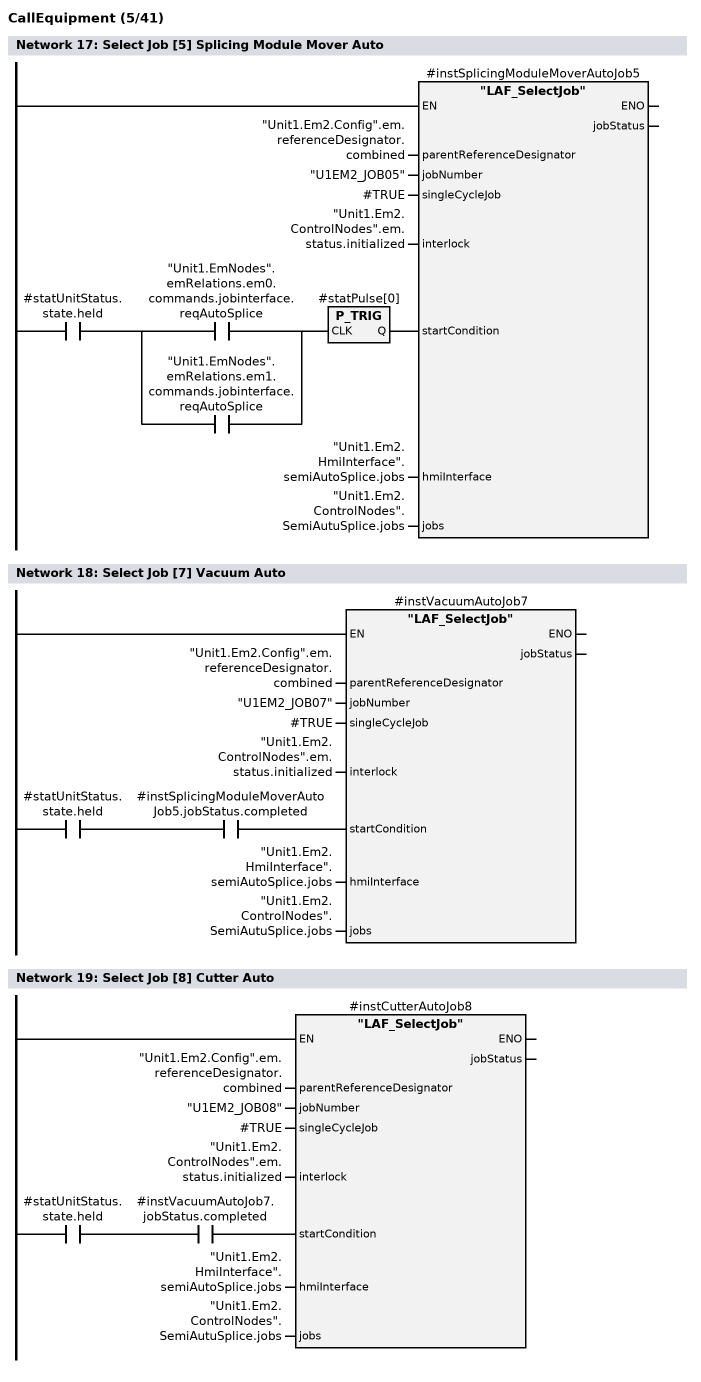
   RUNG wire#powerrail
      #instSplicingModuleMoverAutoJob5(startCondition := wire#w3, parentReferenceDesignator := "Unit1.Em2.Config".em.referenceDesignator.combined, jobNumber := "U1EM2_JOB05", singleCycleJob := #TRUE, interlock := "Unit1.Em2.ControlNodes".em.status.initialized, hmiInterface := "Unit1.Em2.HmiInterface".semiAutoSplice.jobs, jobs := "Unit1.Em2.ControlNodes".SemiAutuSplice.jobs, jobStatus =>)
   END_RUNG
   RUNG wire#powerrail
      Contact( #statUnitStatus.state.held )
      wire#w1
      Contact( "Unit1.EmNodes".emRelations.em0.commands.jobinterface.reqAutoSplice )
      wire#w2
      P_Trig( #statPulse[0] )
   END_RUNG wire#w3
   RUNG wire#w1
      Contact( "Unit1.EmNodes".emRelations.em1.commands.jobinterface.reqAutoSplice )
   END_RUNG wire#w2
   // the same network as SCL:
   #_w1 := #statUnitStatus.state.held AND ("Unit1.EmNodes".emRelations.em0.commands.jobinterface.reqAutoSplice OR "Unit1.EmNodes".emRelations.em1.commands.jobinterface.reqAutoSplice);
   #_w2 := #_w1 AND NOT #statPulse[0];   // rising edge
   #statPulse[0] := #_w1;
   #instSplicingModuleMoverAutoJob5(parentReferenceDesignator := "Unit1.Em2.Config".em.referenceDesignator.combined,   // "LAF_SelectJob"
                           jobNumber := "U1EM2_JOB05",
                           singleCycleJob := #TRUE,
                           interlock := "Unit1.Em2.ControlNodes".em.status.initialized,
                           startCondition := #_w2,
                           hmiInterface := "Unit1.Em2.HmiInterface".semiAutoSplice.jobs,
                           jobs := "Unit1.Em2.ControlNodes".SemiAutuSplice.jobs);
END_REGION

REGION Network 18: Select Job [7] Vacuum Auto
   RUNG wire#powerrail
      #instVacuumAutoJob7(startCondition := wire#w1, parentReferenceDesignator := "Unit1.Em2.Config".em.referenceDesignator.combined, jobNumber := "U1EM2_JOB07", singleCycleJob := #TRUE, interlock := "Unit1.Em2.ControlNodes".em.status.initialized, hmiInterface := "Unit1.Em2.HmiInterface".semiAutoSplice.jobs, jobs := "Unit1.Em2.ControlNodes".SemiAutuSplice.jobs, jobStatus =>)
   END_RUNG
   RUNG wire#powerrail
      Contact( #statUnitStatus.state.held )
      Contact( #instSplicingModuleMoverAutoJob5.jobStatus.completed )
   END_RUNG wire#w1
   // the same network as SCL:
   #instVacuumAutoJob7(parentReferenceDesignator := "Unit1.Em2.Config".em.referenceDesignator.combined,   // "LAF_SelectJob"
                       jobNumber := "U1EM2_JOB07",
                       singleCycleJob := #TRUE,
                       interlock := "Unit1.Em2.ControlNodes".em.status.initialized,
                       startCondition := #statUnitStatus.state.held AND #instSplicingModuleMoverAutoJob5.jobStatus.completed,
                       hmiInterface := "Unit1.Em2.HmiInterface".semiAutoSplice.jobs,
                       jobs := "Unit1.Em2.ControlNodes".SemiAutuSplice.jobs);
END_REGION

REGION Network 19: Select Job [8] Cutter Auto
   RUNG wire#powerrail
      #instCutterAutoJob8(startCondition := wire#w1, parentReferenceDesignator := "Unit1.Em2.Config".em.referenceDesignator.combined, jobNumber := "U1EM2_JOB08", singleCycleJob := #TRUE, interlock := "Unit1.Em2.ControlNodes".em.status.initialized, hmiInterface := "Unit1.Em2.HmiInterface".semiAutoSplice.jobs, jobs := "Unit1.Em2.ControlNodes".SemiAutuSplice.jobs, jobStatus =>)
   END_RUNG
   RUNG wire#powerrail
      Contact( #statUnitStatus.state.held )
      Contact( #instVacuumAutoJob7.jobStatus.completed )
   END_RUNG wire#w1
   // the same network as SCL:
   #instCutterAutoJob8(parentReferenceDesignator := "Unit1.Em2.Config".em.referenceDesignator.combined,   // "LAF_SelectJob"
                       jobNumber := "U1EM2_JOB08",
                       singleCycleJob := #TRUE,
                       interlock := "Unit1.Em2.ControlNodes".em.status.initialized,
                       startCondition := #statUnitStatus.state.held AND #instVacuumAutoJob7.jobStatus.completed,
                       hmiInterface := "Unit1.Em2.HmiInterface".semiAutoSplice.jobs,
                       jobs := "Unit1.Em2.ControlNodes".SemiAutuSplice.jobs);
END_REGION

REGION Network 20: Select Job [9] Left Electrode ReMover Auto
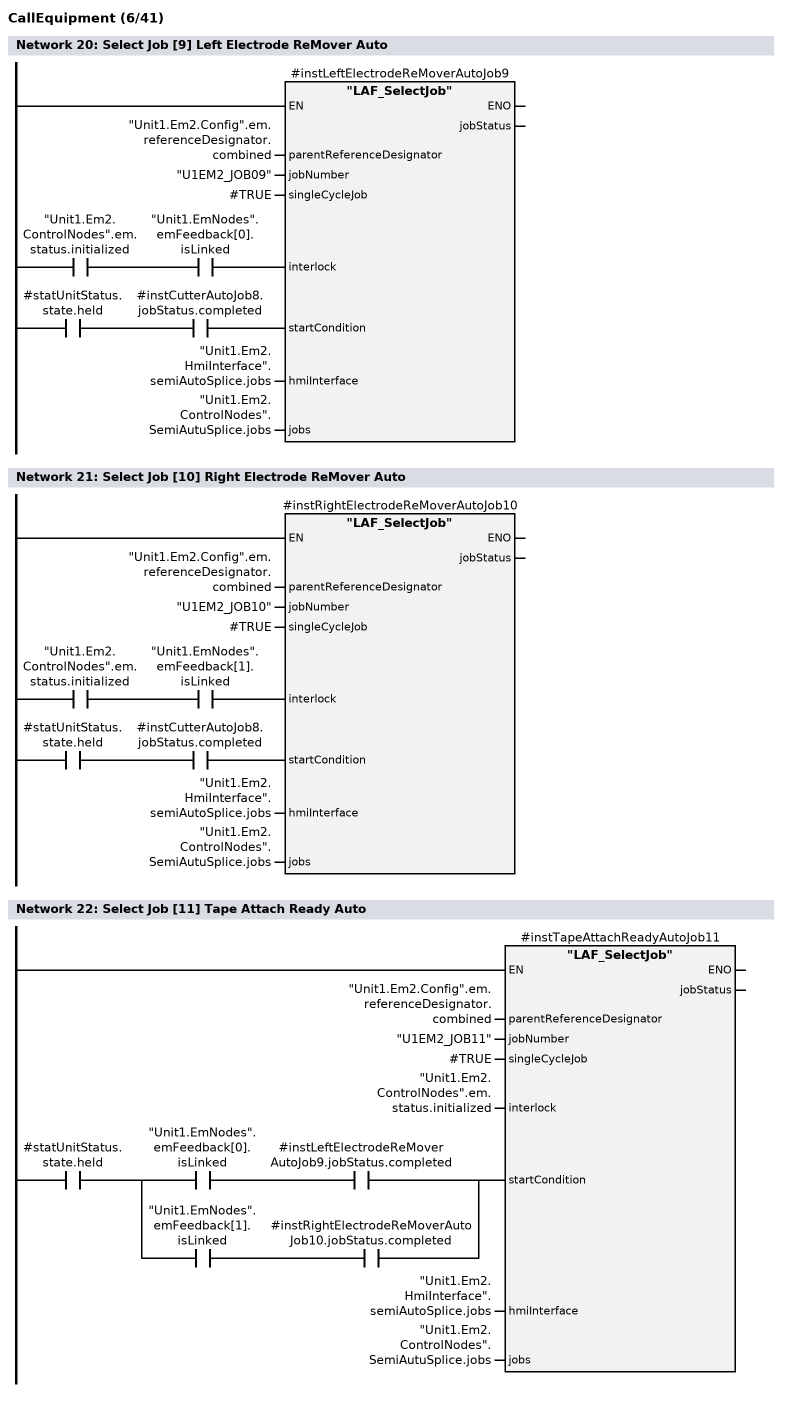
   RUNG wire#powerrail
      #instLeftElectrodeReMoverAutoJob9(interlock := wire#w1, startCondition := wire#w2, parentReferenceDesignator := "Unit1.Em2.Config".em.referenceDesignator.combined, jobNumber := "U1EM2_JOB09", singleCycleJob := #TRUE, hmiInterface := "Unit1.Em2.HmiInterface".semiAutoSplice.jobs, jobs := "Unit1.Em2.ControlNodes".SemiAutuSplice.jobs, jobStatus =>)
   END_RUNG
   RUNG wire#powerrail
      Contact( "Unit1.Em2.ControlNodes".em.status.initialized )
      Contact( "Unit1.EmNodes".emFeedback[0].isLinked )
   END_RUNG wire#w1
   RUNG wire#powerrail
      Contact( #statUnitStatus.state.held )
      Contact( #instCutterAutoJob8.jobStatus.completed )
   END_RUNG wire#w2
   // the same network as SCL:
   #instLeftElectrodeReMoverAutoJob9(parentReferenceDesignator := "Unit1.Em2.Config".em.referenceDesignator.combined,   // "LAF_SelectJob"
                           jobNumber := "U1EM2_JOB09",
                           singleCycleJob := #TRUE,
                           interlock := "Unit1.Em2.ControlNodes".em.status.initialized AND "Unit1.EmNodes".emFeedback[0].isLinked,
                           startCondition := #statUnitStatus.state.held AND #instCutterAutoJob8.jobStatus.completed,
                           hmiInterface := "Unit1.Em2.HmiInterface".semiAutoSplice.jobs,
                           jobs := "Unit1.Em2.ControlNodes".SemiAutuSplice.jobs);
END_REGION

REGION Network 21: Select Job [10] Right Electrode ReMover Auto
   RUNG wire#powerrail
      #instRightElectrodeReMoverAutoJob10(interlock := wire#w1, startCondition := wire#w2, parentReferenceDesignator := "Unit1.Em2.Config".em.referenceDesignator.combined, jobNumber := "U1EM2_JOB10", singleCycleJob := #TRUE, hmiInterface := "Unit1.Em2.HmiInterface".semiAutoSplice.jobs, jobs := "Unit1.Em2.ControlNodes".SemiAutuSplice.jobs, jobStatus =>)
   END_RUNG
   RUNG wire#powerrail
      Contact( "Unit1.Em2.ControlNodes".em.status.initialized )
      Contact( "Unit1.EmNodes".emFeedback[1].isLinked )
   END_RUNG wire#w1
   RUNG wire#powerrail
      Contact( #statUnitStatus.state.held )
      Contact( #instCutterAutoJob8.jobStatus.completed )
   END_RUNG wire#w2
   // the same network as SCL:
   #instRightElectrodeReMoverAutoJob10(parentReferenceDesignator := "Unit1.Em2.Config".em.referenceDesignator.combined,   // "LAF_SelectJob"
                           jobNumber := "U1EM2_JOB10",
                           singleCycleJob := #TRUE,
                           interlock := "Unit1.Em2.ControlNodes".em.status.initialized AND "Unit1.EmNodes".emFeedback[1].isLinked,
                           startCondition := #statUnitStatus.state.held AND #instCutterAutoJob8.jobStatus.completed,
                           hmiInterface := "Unit1.Em2.HmiInterface".semiAutoSplice.jobs,
                           jobs := "Unit1.Em2.ControlNodes".SemiAutuSplice.jobs);
END_REGION

REGION Network 22: Select Job [11] Tape Attach Ready Auto
   RUNG wire#powerrail
      #instTapeAttachReadyAutoJob11(startCondition := wire#w2, parentReferenceDesignator := "Unit1.Em2.Config".em.referenceDesignator.combined, jobNumber := "U1EM2_JOB11", singleCycleJob := #TRUE, interlock := "Unit1.Em2.ControlNodes".em.status.initialized, hmiInterface := "Unit1.Em2.HmiInterface".semiAutoSplice.jobs, jobs := "Unit1.Em2.ControlNodes".SemiAutuSplice.jobs, jobStatus =>)
   END_RUNG
   RUNG wire#powerrail
      Contact( #statUnitStatus.state.held )
      wire#w1
      Contact( "Unit1.EmNodes".emFeedback[0].isLinked )
      Contact( #instLeftElectrodeReMoverAutoJob9.jobStatus.completed )
   END_RUNG wire#w2
   RUNG wire#w1
      Contact( "Unit1.EmNodes".emFeedback[1].isLinked )
      Contact( #instRightElectrodeReMoverAutoJob10.jobStatus.completed )
   END_RUNG wire#w2
   // the same network as SCL:
   #instTapeAttachReadyAutoJob11(parentReferenceDesignator := "Unit1.Em2.Config".em.referenceDesignator.combined,   // "LAF_SelectJob"
                           jobNumber := "U1EM2_JOB11",
                           singleCycleJob := #TRUE,
                           interlock := "Unit1.Em2.ControlNodes".em.status.initialized,
                           startCondition := #statUnitStatus.state.held AND (("Unit1.EmNodes".emFeedback[0].isLinked AND #instLeftElectrodeReMoverAutoJob9.jobStatus.completed) OR ("Unit1.EmNodes".emFeedback[1].isLinked AND #instRightElectrodeReMoverAutoJob10.jobStatus.completed)),
                           hmiInterface := "Unit1.Em2.HmiInterface".semiAutoSplice.jobs,
                           jobs := "Unit1.Em2.ControlNodes".SemiAutuSplice.jobs);
END_REGION

REGION Network 23: Select Job [12] Tape Attach Start Auto
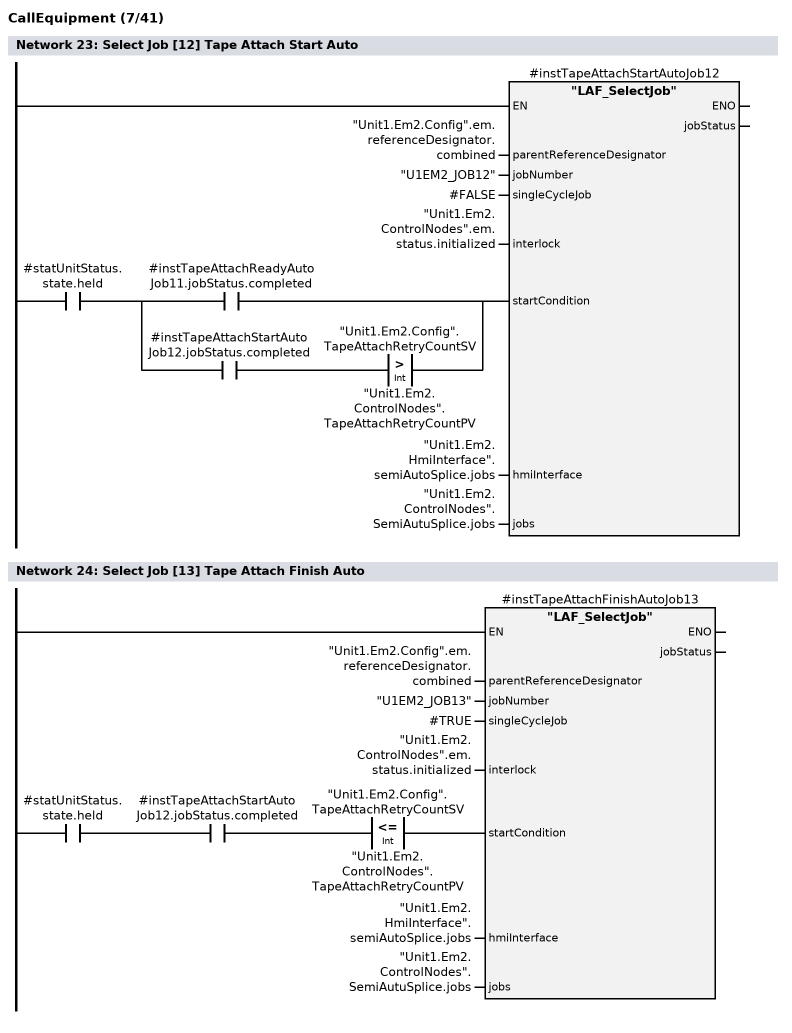
   RUNG wire#powerrail
      #instTapeAttachStartAutoJob12(startCondition := wire#w2, parentReferenceDesignator := "Unit1.Em2.Config".em.referenceDesignator.combined, jobNumber := "U1EM2_JOB12", singleCycleJob := #FALSE, interlock := "Unit1.Em2.ControlNodes".em.status.initialized, hmiInterface := "Unit1.Em2.HmiInterface".semiAutoSplice.jobs, jobs := "Unit1.Em2.ControlNodes".SemiAutuSplice.jobs, jobStatus =>)
   END_RUNG
   RUNG wire#powerrail
      Contact( #statUnitStatus.state.held )
      wire#w1
      Contact( #instTapeAttachReadyAutoJob11.jobStatus.completed )
   END_RUNG wire#w2
   RUNG wire#w1
      Contact( #instTapeAttachStartAutoJob12.jobStatus.completed )
      { S7_Templates := "SrcType := Int" } GT_Contact(in1 := "Unit1.Em2.Config".TapeAttachRetryCountSV, in2 := "Unit1.Em2.ControlNodes".TapeAttachRetryCountPV)
   END_RUNG wire#w2
   // the same network as SCL:
   #instTapeAttachStartAutoJob12(parentReferenceDesignator := "Unit1.Em2.Config".em.referenceDesignator.combined,   // "LAF_SelectJob"
                           jobNumber := "U1EM2_JOB12",
                           singleCycleJob := #FALSE,
                           interlock := "Unit1.Em2.ControlNodes".em.status.initialized,
                           startCondition := #statUnitStatus.state.held AND (#instTapeAttachReadyAutoJob11.jobStatus.completed OR (#instTapeAttachStartAutoJob12.jobStatus.completed AND ("Unit1.Em2.Config".TapeAttachRetryCountSV > "Unit1.Em2.ControlNodes".TapeAttachRetryCountPV))),
                           hmiInterface := "Unit1.Em2.HmiInterface".semiAutoSplice.jobs,
                           jobs := "Unit1.Em2.ControlNodes".SemiAutuSplice.jobs);
END_REGION

REGION Network 24: Select Job [13] Tape Attach Finish Auto
   RUNG wire#powerrail
      #instTapeAttachFinishAutoJob13(startCondition := wire#w1, parentReferenceDesignator := "Unit1.Em2.Config".em.referenceDesignator.combined, jobNumber := "U1EM2_JOB13", singleCycleJob := #TRUE, interlock := "Unit1.Em2.ControlNodes".em.status.initialized, hmiInterface := "Unit1.Em2.HmiInterface".semiAutoSplice.jobs, jobs := "Unit1.Em2.ControlNodes".SemiAutuSplice.jobs, jobStatus =>)
   END_RUNG
   RUNG wire#powerrail
      Contact( #statUnitStatus.state.held )
      Contact( #instTapeAttachStartAutoJob12.jobStatus.completed )
      { S7_Templates := "SrcType := Int" } LE_Contact(in1 := "Unit1.Em2.Config".TapeAttachRetryCountSV, in2 := "Unit1.Em2.ControlNodes".TapeAttachRetryCountPV)
   END_RUNG wire#w1
   // the same network as SCL:
   #instTapeAttachFinishAutoJob13(parentReferenceDesignator := "Unit1.Em2.Config".em.referenceDesignator.combined,   // "LAF_SelectJob"
                           jobNumber := "U1EM2_JOB13",
                           singleCycleJob := #TRUE,
                           interlock := "Unit1.Em2.ControlNodes".em.status.initialized,
                           startCondition := #statUnitStatus.state.held AND #instTapeAttachStartAutoJob12.jobStatus.completed AND ("Unit1.Em2.Config".TapeAttachRetryCountSV <= "Unit1.Em2.ControlNodes".TapeAttachRetryCountPV),
                           hmiInterface := "Unit1.Em2.HmiInterface".semiAutoSplice.jobs,
                           jobs := "Unit1.Em2.ControlNodes".SemiAutuSplice.jobs);
END_REGION

REGION Network 25: Select Job [14] Left Splicing Module Mover Auto
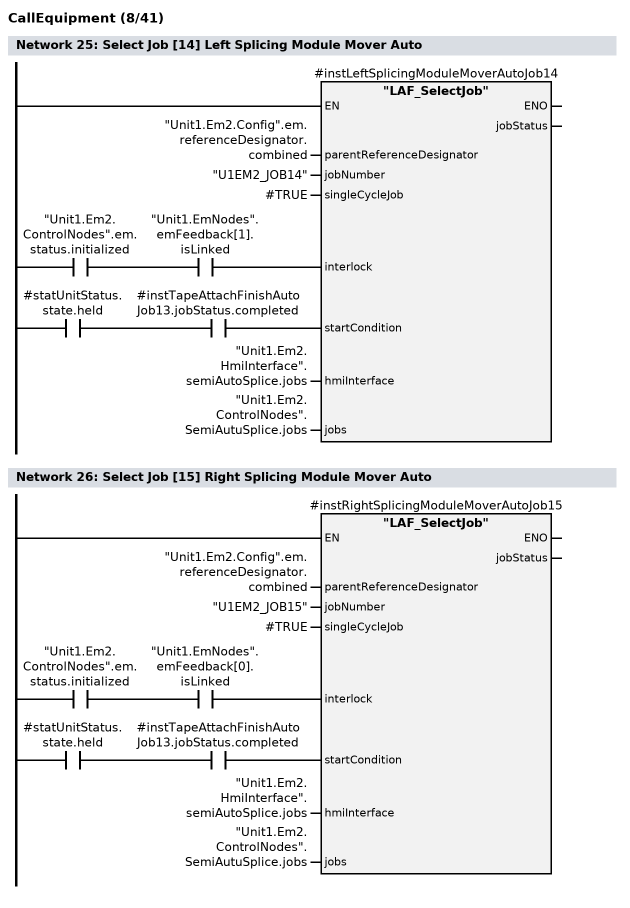
   RUNG wire#powerrail
      #instLeftSplicingModuleMoverAutoJob14(interlock := wire#w1, startCondition := wire#w2, parentReferenceDesignator := "Unit1.Em2.Config".em.referenceDesignator.combined, jobNumber := "U1EM2_JOB14", singleCycleJob := #TRUE, hmiInterface := "Unit1.Em2.HmiInterface".semiAutoSplice.jobs, jobs := "Unit1.Em2.ControlNodes".SemiAutuSplice.jobs, jobStatus =>)
   END_RUNG
   RUNG wire#powerrail
      Contact( "Unit1.Em2.ControlNodes".em.status.initialized )
      Contact( "Unit1.EmNodes".emFeedback[1].isLinked )
   END_RUNG wire#w1
   RUNG wire#powerrail
      Contact( #statUnitStatus.state.held )
      Contact( #instTapeAttachFinishAutoJob13.jobStatus.completed )
   END_RUNG wire#w2
   // the same network as SCL:
   #instLeftSplicingModuleMoverAutoJob14(parentReferenceDesignator := "Unit1.Em2.Config".em.referenceDesignator.combined,   // "LAF_SelectJob"
                           jobNumber := "U1EM2_JOB14",
                           singleCycleJob := #TRUE,
                           interlock := "Unit1.Em2.ControlNodes".em.status.initialized AND "Unit1.EmNodes".emFeedback[1].isLinked,
                           startCondition := #statUnitStatus.state.held AND #instTapeAttachFinishAutoJob13.jobStatus.completed,
                           hmiInterface := "Unit1.Em2.HmiInterface".semiAutoSplice.jobs,
                           jobs := "Unit1.Em2.ControlNodes".SemiAutuSplice.jobs);
END_REGION

REGION Network 26: Select Job [15] Right Splicing Module Mover Auto
   RUNG wire#powerrail
      #instRightSplicingModuleMoverAutoJob15(interlock := wire#w1, startCondition := wire#w2, parentReferenceDesignator := "Unit1.Em2.Config".em.referenceDesignator.combined, jobNumber := "U1EM2_JOB15", singleCycleJob := #TRUE, hmiInterface := "Unit1.Em2.HmiInterface".semiAutoSplice.jobs, jobs := "Unit1.Em2.ControlNodes".SemiAutuSplice.jobs, jobStatus =>)
   END_RUNG
   RUNG wire#powerrail
      Contact( "Unit1.Em2.ControlNodes".em.status.initialized )
      Contact( "Unit1.EmNodes".emFeedback[0].isLinked )
   END_RUNG wire#w1
   RUNG wire#powerrail
      Contact( #statUnitStatus.state.held )
      Contact( #instTapeAttachFinishAutoJob13.jobStatus.completed )
   END_RUNG wire#w2
   // the same network as SCL:
   #instRightSplicingModuleMoverAutoJob15(parentReferenceDesignator := "Unit1.Em2.Config".em.referenceDesignator.combined,   // "LAF_SelectJob"
                           jobNumber := "U1EM2_JOB15",
                           singleCycleJob := #TRUE,
                           interlock := "Unit1.Em2.ControlNodes".em.status.initialized AND "Unit1.EmNodes".emFeedback[0].isLinked,
                           startCondition := #statUnitStatus.state.held AND #instTapeAttachFinishAutoJob13.jobStatus.completed,
                           hmiInterface := "Unit1.Em2.HmiInterface".semiAutoSplice.jobs,
                           jobs := "Unit1.Em2.ControlNodes".SemiAutuSplice.jobs);
END_REGION

REGION Network 27: Select Job [20] Semi Auto Splice Full Auto
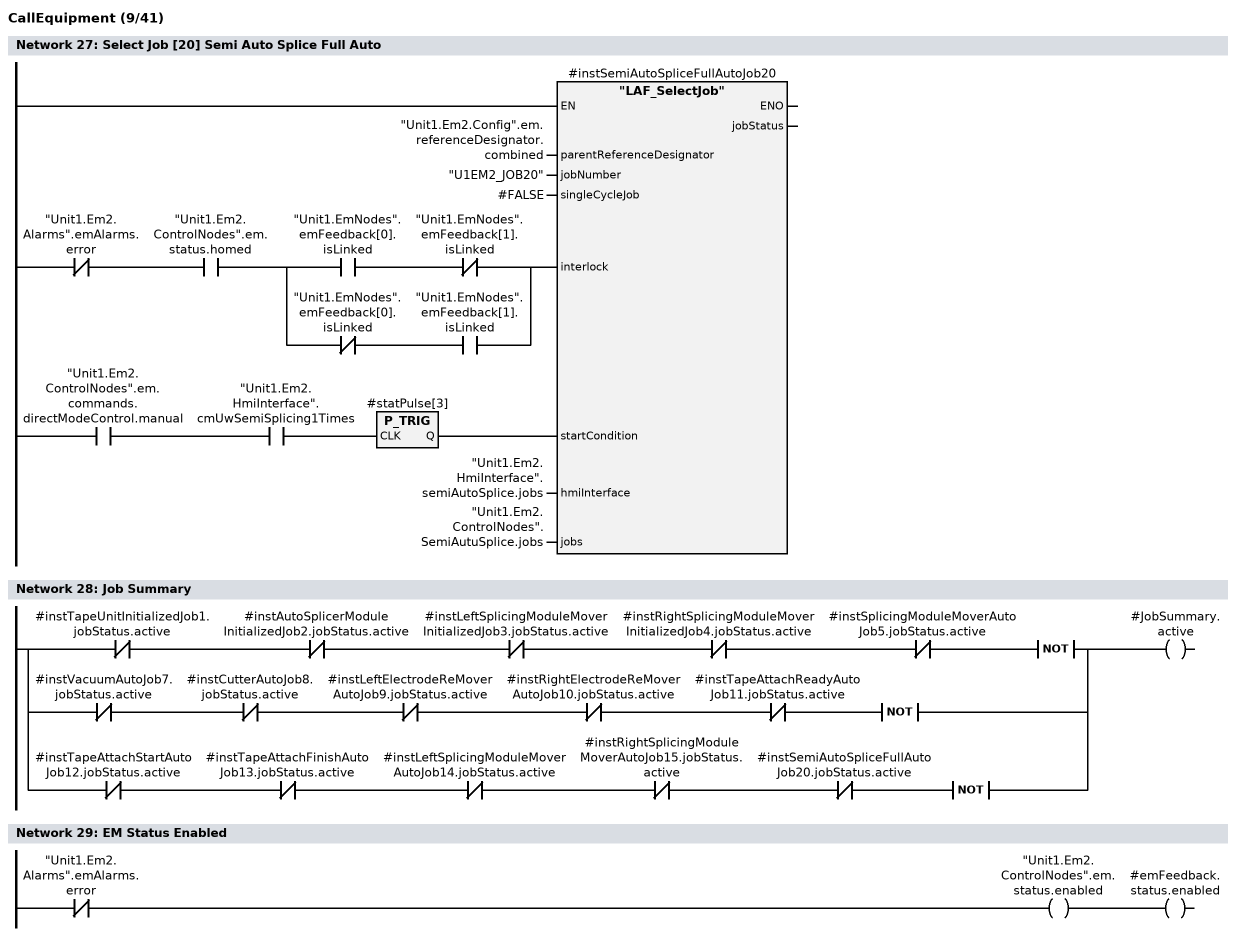
   RUNG wire#powerrail
      #instSemiAutoSpliceFullAutoJob20(interlock := wire#w2, startCondition := wire#w3, parentReferenceDesignator := "Unit1.Em2.Config".em.referenceDesignator.combined, jobNumber := "U1EM2_JOB20", singleCycleJob := #FALSE, hmiInterface := "Unit1.Em2.HmiInterface".semiAutoSplice.jobs, jobs := "Unit1.Em2.ControlNodes".SemiAutuSplice.jobs, jobStatus =>)
   END_RUNG
   RUNG wire#powerrail
      I_Contact( "Unit1.Em2.Alarms".emAlarms.error )
      Contact( "Unit1.Em2.ControlNodes".em.status.homed )
      wire#w1
      Contact( "Unit1.EmNodes".emFeedback[0].isLinked )
      I_Contact( "Unit1.EmNodes".emFeedback[1].isLinked )
   END_RUNG wire#w2
   RUNG wire#w1
      I_Contact( "Unit1.EmNodes".emFeedback[0].isLinked )
      Contact( "Unit1.EmNodes".emFeedback[1].isLinked )
   END_RUNG wire#w2
   RUNG wire#powerrail
      Contact( "Unit1.Em2.ControlNodes".em.commands.directModeControl.manual )
      Contact( "Unit1.Em2.HmiInterface".cmUwSemiSplicing1Times )
      P_Trig( #statPulse[3] )
   END_RUNG wire#w3
   // the same network as SCL:
   #_w1 := "Unit1.Em2.ControlNodes".em.commands.directModeControl.manual AND "Unit1.Em2.HmiInterface".cmUwSemiSplicing1Times;
   #_w2 := #_w1 AND NOT #statPulse[3];   // rising edge
   #statPulse[3] := #_w1;
   #instSemiAutoSpliceFullAutoJob20(parentReferenceDesignator := "Unit1.Em2.Config".em.referenceDesignator.combined,   // "LAF_SelectJob"
                           jobNumber := "U1EM2_JOB20",
                           singleCycleJob := #FALSE,
                           interlock := NOT "Unit1.Em2.Alarms".emAlarms.error AND "Unit1.Em2.ControlNodes".em.status.homed AND (("Unit1.EmNodes".emFeedback[0].isLinked AND NOT "Unit1.EmNodes".emFeedback[1].isLinked) OR (NOT "Unit1.EmNodes".emFeedback[0].isLinked AND "Unit1.EmNodes".emFeedback[1].isLinked)),
                           startCondition := #_w2,
                           hmiInterface := "Unit1.Em2.HmiInterface".semiAutoSplice.jobs,
                           jobs := "Unit1.Em2.ControlNodes".SemiAutuSplice.jobs);
END_REGION

REGION Network 28: Job Summary
   RUNG wire#powerrail
      I_Contact( #instTapeUnitInitializedJob1.jobStatus.active )
      I_Contact( #instAutoSplicerModuleInitializedJob2.jobStatus.active )
      I_Contact( #instLeftSplicingModuleMoverInitializedJob3.jobStatus.active )
      I_Contact( #instRightSplicingModuleMoverInitializedJob4.jobStatus.active )
      I_Contact( #instSplicingModuleMoverAutoJob5.jobStatus.active )
      Not()
      wire#w1
      Coil( #JobSummary.active )
   END_RUNG
   RUNG wire#powerrail
      I_Contact( #instVacuumAutoJob7.jobStatus.active )
      I_Contact( #instCutterAutoJob8.jobStatus.active )
      I_Contact( #instLeftElectrodeReMoverAutoJob9.jobStatus.active )
      I_Contact( #instRightElectrodeReMoverAutoJob10.jobStatus.active )
      I_Contact( #instTapeAttachReadyAutoJob11.jobStatus.active )
      Not()
   END_RUNG wire#w1
   RUNG wire#powerrail
      I_Contact( #instTapeAttachStartAutoJob12.jobStatus.active )
      I_Contact( #instTapeAttachFinishAutoJob13.jobStatus.active )
      I_Contact( #instLeftSplicingModuleMoverAutoJob14.jobStatus.active )
      I_Contact( #instRightSplicingModuleMoverAutoJob15.jobStatus.active )
      I_Contact( #instSemiAutoSpliceFullAutoJob20.jobStatus.active )
      Not()
   END_RUNG wire#w1
   // the same network as SCL:
   #JobSummary.active := NOT (NOT #instTapeUnitInitializedJob1.jobStatus.active AND NOT #instAutoSplicerModuleInitializedJob2.jobStatus.active AND NOT #instLeftSplicingModuleMoverInitializedJob3.jobStatus.active AND NOT #instRightSplicingModuleMoverInitializedJob4.jobStatus.active AND NOT #instSplicingModuleMoverAutoJob5.jobStatus.active) OR NOT (NOT #instVacuumAutoJob7.jobStatus.active AND NOT #instCutterAutoJob8.jobStatus.active AND NOT #instLeftElectrodeReMoverAutoJob9.jobStatus.active AND NOT #instRightElectrodeReMoverAutoJob10.jobStatus.active AND NOT #instTapeAttachReadyAutoJob11.jobStatus.active) OR NOT (NOT #instTapeAttachStartAutoJob12.jobStatus.active AND NOT #instTapeAttachFinishAutoJob13.jobStatus.active AND NOT #instLeftSplicingModuleMoverAutoJob14.jobStatus.active AND NOT #instRightSplicingModuleMoverAutoJob15.jobStatus.active AND NOT #instSemiAutoSpliceFullAutoJob20.jobStatus.active);
END_REGION

REGION Network 29: EM Status Enabled
   RUNG wire#powerrail
      I_Contact( "Unit1.Em2.Alarms".emAlarms.error )
      Coil( "Unit1.Em2.ControlNodes".em.status.enabled )
      Coil( #emFeedback.status.enabled )
   END_RUNG
   // the same network as SCL:
   "Unit1.Em2.ControlNodes".em.status.enabled := NOT "Unit1.Em2.Alarms".emAlarms.error;
   #emFeedback.status.enabled := NOT "Unit1.Em2.Alarms".emAlarms.error;
END_REGION

REGION Network 30: EM Status initialized
   // Set em to initialized here. Usually this is done when the initialization job is completed.
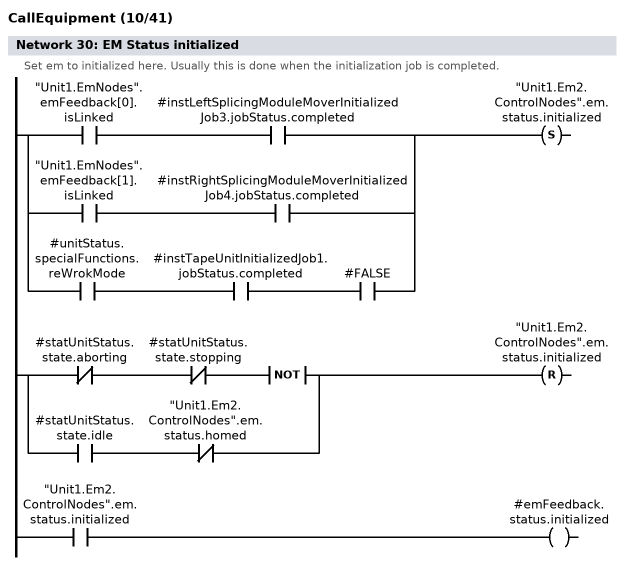
   RUNG wire#powerrail
      Contact( "Unit1.EmNodes".emFeedback[0].isLinked )
      Contact( #instLeftSplicingModuleMoverInitializedJob3.jobStatus.completed )
      wire#w1
      S_Coil( "Unit1.Em2.ControlNodes".em.status.initialized )
   END_RUNG
   RUNG wire#powerrail
      Contact( "Unit1.EmNodes".emFeedback[1].isLinked )
      Contact( #instRightSplicingModuleMoverInitializedJob4.jobStatus.completed )
   END_RUNG wire#w1
   RUNG wire#powerrail
      Contact( #unitStatus.specialFunctions.reWrokMode )
      Contact( #instTapeUnitInitializedJob1.jobStatus.completed )
      Contact( #FALSE )
   END_RUNG wire#w1
   RUNG wire#powerrail
      I_Contact( #statUnitStatus.state.aborting )
      I_Contact( #statUnitStatus.state.stopping )
      Not()
      wire#w2
      R_Coil( "Unit1.Em2.ControlNodes".em.status.initialized )
   END_RUNG
   RUNG wire#powerrail
      Contact( #statUnitStatus.state.idle )
      I_Contact( "Unit1.Em2.ControlNodes".em.status.homed )
   END_RUNG wire#w2
   RUNG wire#powerrail
      Contact( "Unit1.Em2.ControlNodes".em.status.initialized )
      Coil( #emFeedback.status.initialized )
   END_RUNG
   // the same network as SCL:
   IF ("Unit1.EmNodes".emFeedback[0].isLinked AND #instLeftSplicingModuleMoverInitializedJob3.jobStatus.completed) OR ("Unit1.EmNodes".emFeedback[1].isLinked AND #instRightSplicingModuleMoverInitializedJob4.jobStatus.completed) OR (#unitStatus.specialFunctions.reWrokMode AND #instTapeUnitInitializedJob1.jobStatus.completed AND #FALSE) THEN
       "Unit1.Em2.ControlNodes".em.status.initialized := TRUE;
   END_IF;
   IF NOT (NOT #statUnitStatus.state.aborting AND NOT #statUnitStatus.state.stopping) OR (#statUnitStatus.state.idle AND NOT "Unit1.Em2.ControlNodes".em.status.homed) THEN
       "Unit1.Em2.ControlNodes".em.status.initialized := FALSE;
   END_IF;
   #emFeedback.status.initialized := "Unit1.Em2.ControlNodes".em.status.initialized;
END_REGION

REGION Network 31: EM Status Homed
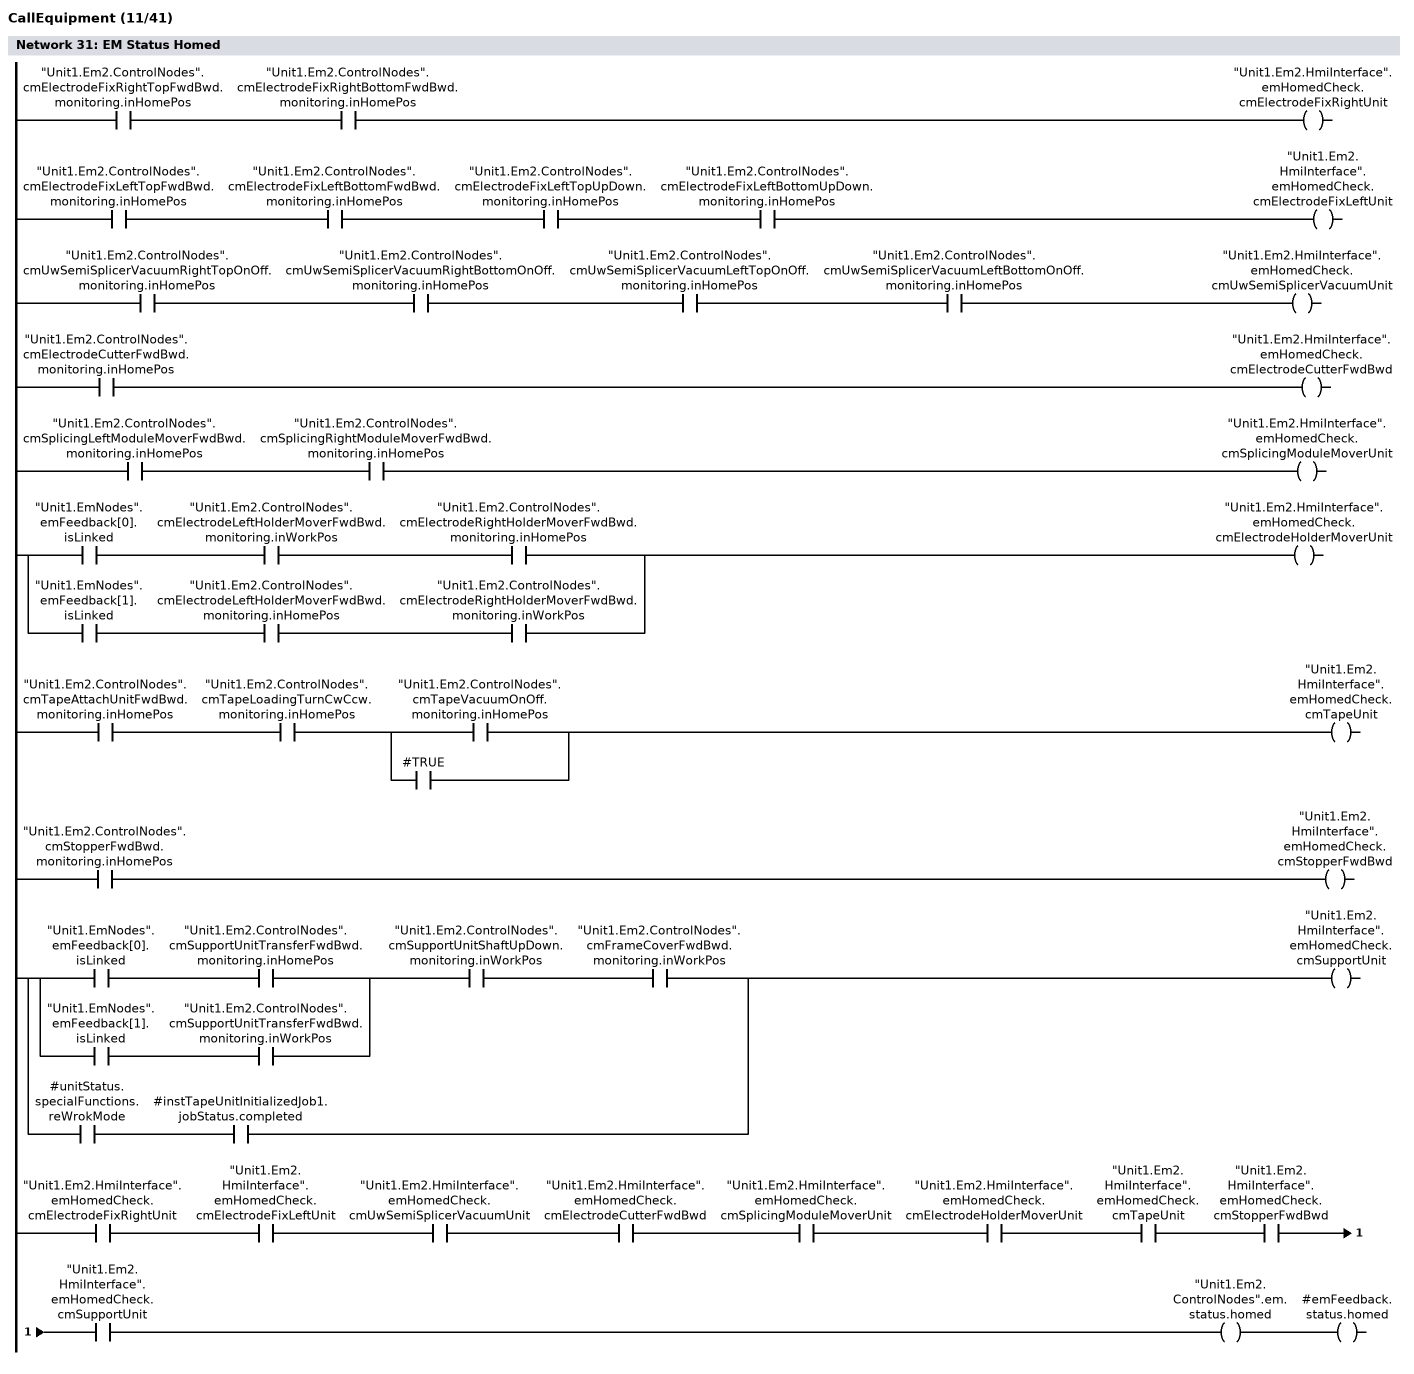
   RUNG wire#powerrail
      Contact( "Unit1.Em2.ControlNodes".cmElectrodeFixRightTopFwdBwd.monitoring.inHomePos )
      Contact( "Unit1.Em2.ControlNodes".cmElectrodeFixRightBottomFwdBwd.monitoring.inHomePos )
      Coil( "Unit1.Em2.HmiInterface".emHomedCheck.cmElectrodeFixRightUnit )
   END_RUNG
   RUNG wire#powerrail
      Contact( "Unit1.Em2.ControlNodes".cmElectrodeFixLeftTopFwdBwd.monitoring.inHomePos )
      Contact( "Unit1.Em2.ControlNodes".cmElectrodeFixLeftBottomFwdBwd.monitoring.inHomePos )
      Contact( "Unit1.Em2.ControlNodes".cmElectrodeFixLeftTopUpDown.monitoring.inHomePos )
      Contact( "Unit1.Em2.ControlNodes".cmElectrodeFixLeftBottomUpDown.monitoring.inHomePos )
      Coil( "Unit1.Em2.HmiInterface".emHomedCheck.cmElectrodeFixLeftUnit )
   END_RUNG
   RUNG wire#powerrail
      Contact( "Unit1.Em2.ControlNodes".cmUwSemiSplicerVacuumRightTopOnOff.monitoring.inHomePos )
      Contact( "Unit1.Em2.ControlNodes".cmUwSemiSplicerVacuumRightBottomOnOff.monitoring.inHomePos )
      Contact( "Unit1.Em2.ControlNodes".cmUwSemiSplicerVacuumLeftTopOnOff.monitoring.inHomePos )
      Contact( "Unit1.Em2.ControlNodes".cmUwSemiSplicerVacuumLeftBottomOnOff.monitoring.inHomePos )
      Coil( "Unit1.Em2.HmiInterface".emHomedCheck.cmUwSemiSplicerVacuumUnit )
   END_RUNG
   RUNG wire#powerrail
      Contact( "Unit1.Em2.ControlNodes".cmElectrodeCutterFwdBwd.monitoring.inHomePos )
      Coil( "Unit1.Em2.HmiInterface".emHomedCheck.cmElectrodeCutterFwdBwd )
   END_RUNG
   RUNG wire#powerrail
      Contact( "Unit1.Em2.ControlNodes".cmSplicingLeftModuleMoverFwdBwd.monitoring.inHomePos )
      Contact( "Unit1.Em2.ControlNodes".cmSplicingRightModuleMoverFwdBwd.monitoring.inHomePos )
      Coil( "Unit1.Em2.HmiInterface".emHomedCheck.cmSplicingModuleMoverUnit )
   END_RUNG
   RUNG wire#powerrail
      Contact( "Unit1.EmNodes".emFeedback[0].isLinked )
      Contact( "Unit1.Em2.ControlNodes".cmElectrodeLeftHolderMoverFwdBwd.monitoring.inWorkPos )
      Contact( "Unit1.Em2.ControlNodes".cmElectrodeRightHolderMoverFwdBwd.monitoring.inHomePos )
      wire#w1
      Coil( "Unit1.Em2.HmiInterface".emHomedCheck.cmElectrodeHolderMoverUnit )
   END_RUNG
   RUNG wire#powerrail
      Contact( "Unit1.EmNodes".emFeedback[1].isLinked )
      Contact( "Unit1.Em2.ControlNodes".cmElectrodeLeftHolderMoverFwdBwd.monitoring.inHomePos )
      Contact( "Unit1.Em2.ControlNodes".cmElectrodeRightHolderMoverFwdBwd.monitoring.inWorkPos )
   END_RUNG wire#w1
   RUNG wire#powerrail
      Contact( "Unit1.Em2.ControlNodes".cmTapeAttachUnitFwdBwd.monitoring.inHomePos )
      Contact( "Unit1.Em2.ControlNodes".cmTapeLoadingTurnCwCcw.monitoring.inHomePos )
      wire#w2
      Contact( "Unit1.Em2.ControlNodes".cmTapeVacuumOnOff.monitoring.inHomePos )
      wire#w3
      Coil( "Unit1.Em2.HmiInterface".emHomedCheck.cmTapeUnit )
   END_RUNG
   RUNG wire#w2
      Contact( #TRUE )
   END_RUNG wire#w3
   RUNG wire#powerrail
      Contact( "Unit1.Em2.ControlNodes".cmStopperFwdBwd.monitoring.inHomePos )
      Coil( "Unit1.Em2.HmiInterface".emHomedCheck.cmStopperFwdBwd )
   END_RUNG
   RUNG wire#powerrail
      Contact( "Unit1.EmNodes".emFeedback[0].isLinked )
      Contact( "Unit1.Em2.ControlNodes".cmSupportUnitTransferFwdBwd.monitoring.inHomePos )
      wire#w4
      Contact( "Unit1.Em2.ControlNodes".cmSupportUnitShaftUpDown.monitoring.inWorkPos )
      Contact( "Unit1.Em2.ControlNodes".cmFrameCoverFwdBwd.monitoring.inWorkPos )
      wire#w5
      Coil( "Unit1.Em2.HmiInterface".emHomedCheck.cmSupportUnit )
   END_RUNG
   RUNG wire#powerrail
      Contact( "Unit1.EmNodes".emFeedback[1].isLinked )
      Contact( "Unit1.Em2.ControlNodes".cmSupportUnitTransferFwdBwd.monitoring.inWorkPos )
   END_RUNG wire#w4
   RUNG wire#powerrail
      Contact( #unitStatus.specialFunctions.reWrokMode )
      Contact( #instTapeUnitInitializedJob1.jobStatus.completed )
   END_RUNG wire#w5
   RUNG wire#powerrail
      Contact( "Unit1.Em2.HmiInterface".emHomedCheck.cmElectrodeFixRightUnit )
      Contact( "Unit1.Em2.HmiInterface".emHomedCheck.cmElectrodeFixLeftUnit )
      Contact( "Unit1.Em2.HmiInterface".emHomedCheck.cmUwSemiSplicerVacuumUnit )
      Contact( "Unit1.Em2.HmiInterface".emHomedCheck.cmElectrodeCutterFwdBwd )
      Contact( "Unit1.Em2.HmiInterface".emHomedCheck.cmSplicingModuleMoverUnit )
      Contact( "Unit1.Em2.HmiInterface".emHomedCheck.cmElectrodeHolderMoverUnit )
      Contact( "Unit1.Em2.HmiInterface".emHomedCheck.cmTapeUnit )
      Contact( "Unit1.Em2.HmiInterface".emHomedCheck.cmStopperFwdBwd )
      Contact( "Unit1.Em2.HmiInterface".emHomedCheck.cmSupportUnit )
      Coil( "Unit1.Em2.ControlNodes".em.status.homed )
      Coil( #emFeedback.status.homed )
   END_RUNG
   // the same network as SCL:
   "Unit1.Em2.HmiInterface".emHomedCheck.cmElectrodeFixRightUnit := "Unit1.Em2.ControlNodes".cmElectrodeFixRightTopFwdBwd.monitoring.inHomePos AND "Unit1.Em2.ControlNodes".cmElectrodeFixRightBottomFwdBwd.monitoring.inHomePos;
   "Unit1.Em2.HmiInterface".emHomedCheck.cmElectrodeFixLeftUnit := "Unit1.Em2.ControlNodes".cmElectrodeFixLeftTopFwdBwd.monitoring.inHomePos AND "Unit1.Em2.ControlNodes".cmElectrodeFixLeftBottomFwdBwd.monitoring.inHomePos AND "Unit1.Em2.ControlNodes".cmElectrodeFixLeftTopUpDown.monitoring.inHomePos AND "Unit1.Em2.ControlNodes".cmElectrodeFixLeftBottomUpDown.monitoring.inHomePos;
   "Unit1.Em2.HmiInterface".emHomedCheck.cmUwSemiSplicerVacuumUnit := "Unit1.Em2.ControlNodes".cmUwSemiSplicerVacuumRightTopOnOff.monitoring.inHomePos AND "Unit1.Em2.ControlNodes".cmUwSemiSplicerVacuumRightBottomOnOff.monitoring.inHomePos AND "Unit1.Em2.ControlNodes".cmUwSemiSplicerVacuumLeftTopOnOff.monitoring.inHomePos AND "Unit1.Em2.ControlNodes".cmUwSemiSplicerVacuumLeftBottomOnOff.monitoring.inHomePos;
   "Unit1.Em2.HmiInterface".emHomedCheck.cmElectrodeCutterFwdBwd := "Unit1.Em2.ControlNodes".cmElectrodeCutterFwdBwd.monitoring.inHomePos;
   "Unit1.Em2.HmiInterface".emHomedCheck.cmSplicingModuleMoverUnit := "Unit1.Em2.ControlNodes".cmSplicingLeftModuleMoverFwdBwd.monitoring.inHomePos AND "Unit1.Em2.ControlNodes".cmSplicingRightModuleMoverFwdBwd.monitoring.inHomePos;
   "Unit1.Em2.HmiInterface".emHomedCheck.cmElectrodeHolderMoverUnit := ("Unit1.EmNodes".emFeedback[0].isLinked AND "Unit1.Em2.ControlNodes".cmElectrodeLeftHolderMoverFwdBwd.monitoring.inWorkPos AND "Unit1.Em2.ControlNodes".cmElectrodeRightHolderMoverFwdBwd.monitoring.inHomePos) OR ("Unit1.EmNodes".emFeedback[1].isLinked AND "Unit1.Em2.ControlNodes".cmElectrodeLeftHolderMoverFwdBwd.monitoring.inHomePos AND "Unit1.Em2.ControlNodes".cmElectrodeRightHolderMoverFwdBwd.monitoring.inWorkPos);
   "Unit1.Em2.HmiInterface".emHomedCheck.cmTapeUnit := "Unit1.Em2.ControlNodes".cmTapeAttachUnitFwdBwd.monitoring.inHomePos AND "Unit1.Em2.ControlNodes".cmTapeLoadingTurnCwCcw.monitoring.inHomePos AND ("Unit1.Em2.ControlNodes".cmTapeVacuumOnOff.monitoring.inHomePos OR #TRUE);
   "Unit1.Em2.HmiInterface".emHomedCheck.cmStopperFwdBwd := "Unit1.Em2.ControlNodes".cmStopperFwdBwd.monitoring.inHomePos;
   "Unit1.Em2.HmiInterface".emHomedCheck.cmSupportUnit := ((("Unit1.EmNodes".emFeedback[0].isLinked AND "Unit1.Em2.ControlNodes".cmSupportUnitTransferFwdBwd.monitoring.inHomePos) OR ("Unit1.EmNodes".emFeedback[1].isLinked AND "Unit1.Em2.ControlNodes".cmSupportUnitTransferFwdBwd.monitoring.inWorkPos)) AND "Unit1.Em2.ControlNodes".cmSupportUnitShaftUpDown.monitoring.inWorkPos AND "Unit1.Em2.ControlNodes".cmFrameCoverFwdBwd.monitoring.inWorkPos) OR (#unitStatus.specialFunctions.reWrokMode AND #instTapeUnitInitializedJob1.jobStatus.completed);
   "Unit1.Em2.ControlNodes".em.status.homed := "Unit1.Em2.HmiInterface".emHomedCheck.cmElectrodeFixRightUnit AND "Unit1.Em2.HmiInterface".emHomedCheck.cmElectrodeFixLeftUnit AND "Unit1.Em2.HmiInterface".emHomedCheck.cmUwSemiSplicerVacuumUnit AND "Unit1.Em2.HmiInterface".emHomedCheck.cmElectrodeCutterFwdBwd AND "Unit1.Em2.HmiInterface".emHomedCheck.cmSplicingModuleMoverUnit AND "Unit1.Em2.HmiInterface".emHomedCheck.cmElectrodeHolderMoverUnit AND "Unit1.Em2.HmiInterface".emHomedCheck.cmTapeUnit AND "Unit1.Em2.HmiInterface".emHomedCheck.cmStopperFwdBwd AND "Unit1.Em2.HmiInterface".emHomedCheck.cmSupportUnit;
   #emFeedback.status.homed := "Unit1.Em2.ControlNodes".em.status.homed;
END_REGION

REGION Network 32: Call Sequence [1] Semi Auto Splice
   // Call of the em logic
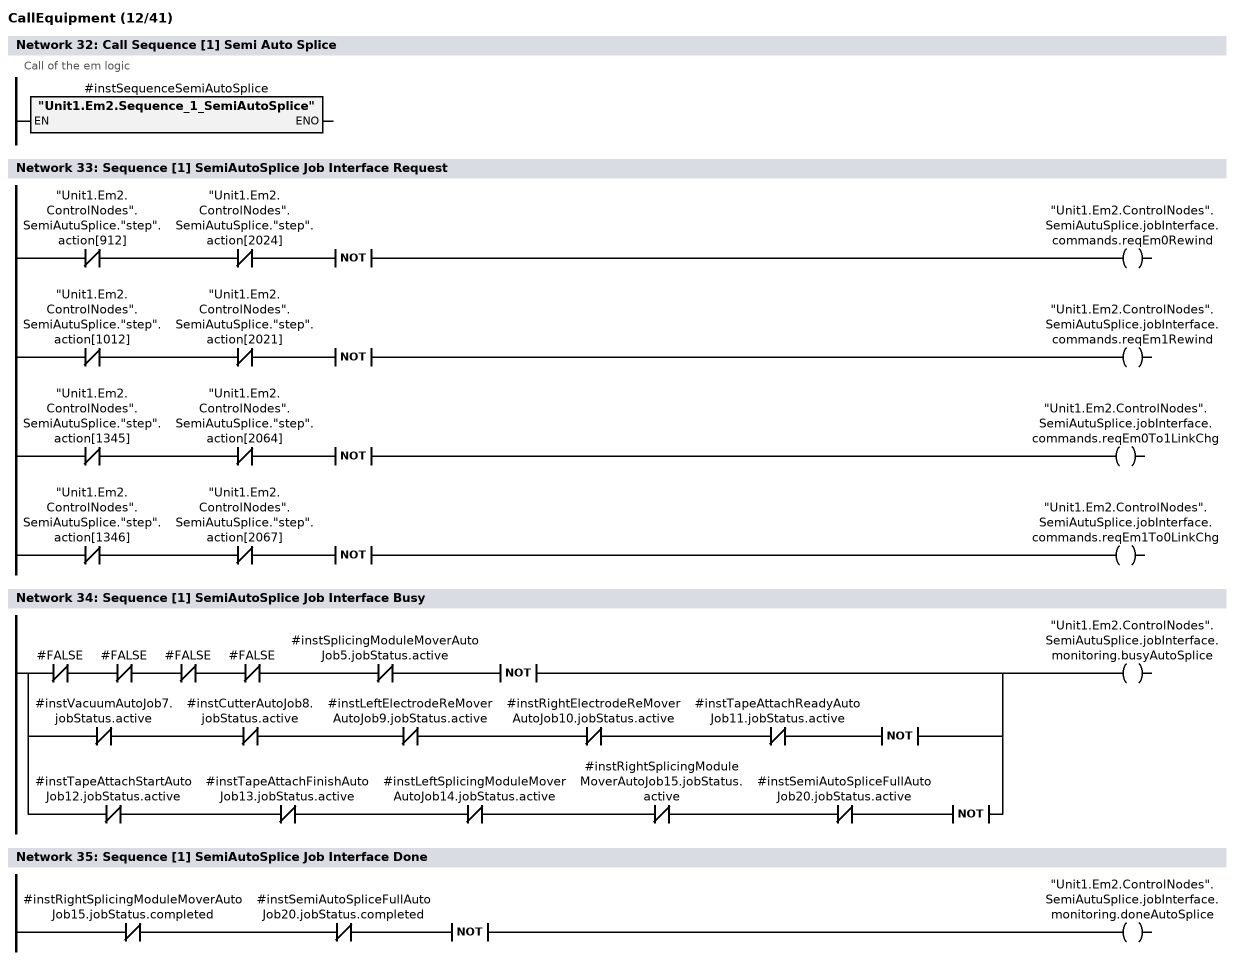
   RUNG wire#powerrail
      #instSequenceSemiAutoSplice()
   END_RUNG
   // the same network as SCL:
   #instSequenceSemiAutoSplice();   // "Unit1.Em2.Sequence_1_SemiAutoSplice"
END_REGION

REGION Network 33: Sequence [1] SemiAutoSplice Job Interface Request
   RUNG wire#powerrail
      I_Contact( "Unit1.Em2.ControlNodes".SemiAutuSplice."step".action[912] )
      I_Contact( "Unit1.Em2.ControlNodes".SemiAutuSplice."step".action[2024] )
      Not()
      Coil( "Unit1.Em2.ControlNodes".SemiAutuSplice.jobInterface.commands.reqEm0Rewind )
   END_RUNG
   RUNG wire#powerrail
      I_Contact( "Unit1.Em2.ControlNodes".SemiAutuSplice."step".action[1012] )
      I_Contact( "Unit1.Em2.ControlNodes".SemiAutuSplice."step".action[2021] )
      Not()
      Coil( "Unit1.Em2.ControlNodes".SemiAutuSplice.jobInterface.commands.reqEm1Rewind )
   END_RUNG
   RUNG wire#powerrail
      I_Contact( "Unit1.Em2.ControlNodes".SemiAutuSplice."step".action[1345] )
      I_Contact( "Unit1.Em2.ControlNodes".SemiAutuSplice."step".action[2064] )
      Not()
      Coil( "Unit1.Em2.ControlNodes".SemiAutuSplice.jobInterface.commands.reqEm0To1LinkChg )
   END_RUNG
   RUNG wire#powerrail
      I_Contact( "Unit1.Em2.ControlNodes".SemiAutuSplice."step".action[1346] )
      I_Contact( "Unit1.Em2.ControlNodes".SemiAutuSplice."step".action[2067] )
      Not()
      Coil( "Unit1.Em2.ControlNodes".SemiAutuSplice.jobInterface.commands.reqEm1To0LinkChg )
   END_RUNG
   // the same network as SCL:
   "Unit1.Em2.ControlNodes".SemiAutuSplice.jobInterface.commands.reqEm0Rewind := NOT (NOT "Unit1.Em2.ControlNodes".SemiAutuSplice."step".action[912] AND NOT "Unit1.Em2.ControlNodes".SemiAutuSplice."step".action[2024]);
   "Unit1.Em2.ControlNodes".SemiAutuSplice.jobInterface.commands.reqEm1Rewind := NOT (NOT "Unit1.Em2.ControlNodes".SemiAutuSplice."step".action[1012] AND NOT "Unit1.Em2.ControlNodes".SemiAutuSplice."step".action[2021]);
   "Unit1.Em2.ControlNodes".SemiAutuSplice.jobInterface.commands.reqEm0To1LinkChg := NOT (NOT "Unit1.Em2.ControlNodes".SemiAutuSplice."step".action[1345] AND NOT "Unit1.Em2.ControlNodes".SemiAutuSplice."step".action[2064]);
   "Unit1.Em2.ControlNodes".SemiAutuSplice.jobInterface.commands.reqEm1To0LinkChg := NOT (NOT "Unit1.Em2.ControlNodes".SemiAutuSplice."step".action[1346] AND NOT "Unit1.Em2.ControlNodes".SemiAutuSplice."step".action[2067]);
END_REGION

REGION Network 34: Sequence [1] SemiAutoSplice Job Interface Busy
   RUNG wire#powerrail
      I_Contact( #FALSE )
      I_Contact( #FALSE )
      I_Contact( #FALSE )
      I_Contact( #FALSE )
      I_Contact( #instSplicingModuleMoverAutoJob5.jobStatus.active )
      Not()
      wire#w1
      Coil( "Unit1.Em2.ControlNodes".SemiAutuSplice.jobInterface.monitoring.busyAutoSplice )
   END_RUNG
   RUNG wire#powerrail
      I_Contact( #instVacuumAutoJob7.jobStatus.active )
      I_Contact( #instCutterAutoJob8.jobStatus.active )
      I_Contact( #instLeftElectrodeReMoverAutoJob9.jobStatus.active )
      I_Contact( #instRightElectrodeReMoverAutoJob10.jobStatus.active )
      I_Contact( #instTapeAttachReadyAutoJob11.jobStatus.active )
      Not()
   END_RUNG wire#w1
   RUNG wire#powerrail
      I_Contact( #instTapeAttachStartAutoJob12.jobStatus.active )
      I_Contact( #instTapeAttachFinishAutoJob13.jobStatus.active )
      I_Contact( #instLeftSplicingModuleMoverAutoJob14.jobStatus.active )
      I_Contact( #instRightSplicingModuleMoverAutoJob15.jobStatus.active )
      I_Contact( #instSemiAutoSpliceFullAutoJob20.jobStatus.active )
      Not()
   END_RUNG wire#w1
   // the same network as SCL:
   "Unit1.Em2.ControlNodes".SemiAutuSplice.jobInterface.monitoring.busyAutoSplice := NOT (NOT #FALSE AND NOT #FALSE AND NOT #FALSE AND NOT #FALSE AND NOT #instSplicingModuleMoverAutoJob5.jobStatus.active) OR NOT (NOT #instVacuumAutoJob7.jobStatus.active AND NOT #instCutterAutoJob8.jobStatus.active AND NOT #instLeftElectrodeReMoverAutoJob9.jobStatus.active AND NOT #instRightElectrodeReMoverAutoJob10.jobStatus.active AND NOT #instTapeAttachReadyAutoJob11.jobStatus.active) OR NOT (NOT #instTapeAttachStartAutoJob12.jobStatus.active AND NOT #instTapeAttachFinishAutoJob13.jobStatus.active AND NOT #instLeftSplicingModuleMoverAutoJob14.jobStatus.active AND NOT #instRightSplicingModuleMoverAutoJob15.jobStatus.active AND NOT #instSemiAutoSpliceFullAutoJob20.jobStatus.active);
END_REGION

REGION Network 35: Sequence [1] SemiAutoSplice Job Interface Done
   RUNG wire#powerrail
      I_Contact( #instRightSplicingModuleMoverAutoJob15.jobStatus.completed )
      I_Contact( #instSemiAutoSpliceFullAutoJob20.jobStatus.completed )
      Not()
      Coil( "Unit1.Em2.ControlNodes".SemiAutuSplice.jobInterface.monitoring.doneAutoSplice )
   END_RUNG
   // the same network as SCL:
   "Unit1.Em2.ControlNodes".SemiAutuSplice.jobInterface.monitoring.doneAutoSplice := NOT (NOT #instRightSplicingModuleMoverAutoJob15.jobStatus.completed AND NOT #instSemiAutoSpliceFullAutoJob20.jobStatus.completed);
END_REGION

REGION Network 36: ******************** Control Modules (TwoWayActuator) ********************
   // Call control modules that are sensors before the em logic (jobs and sequence), so that the latest value is used in the logic.
END_REGION

REGION Network 37: Reset CMS
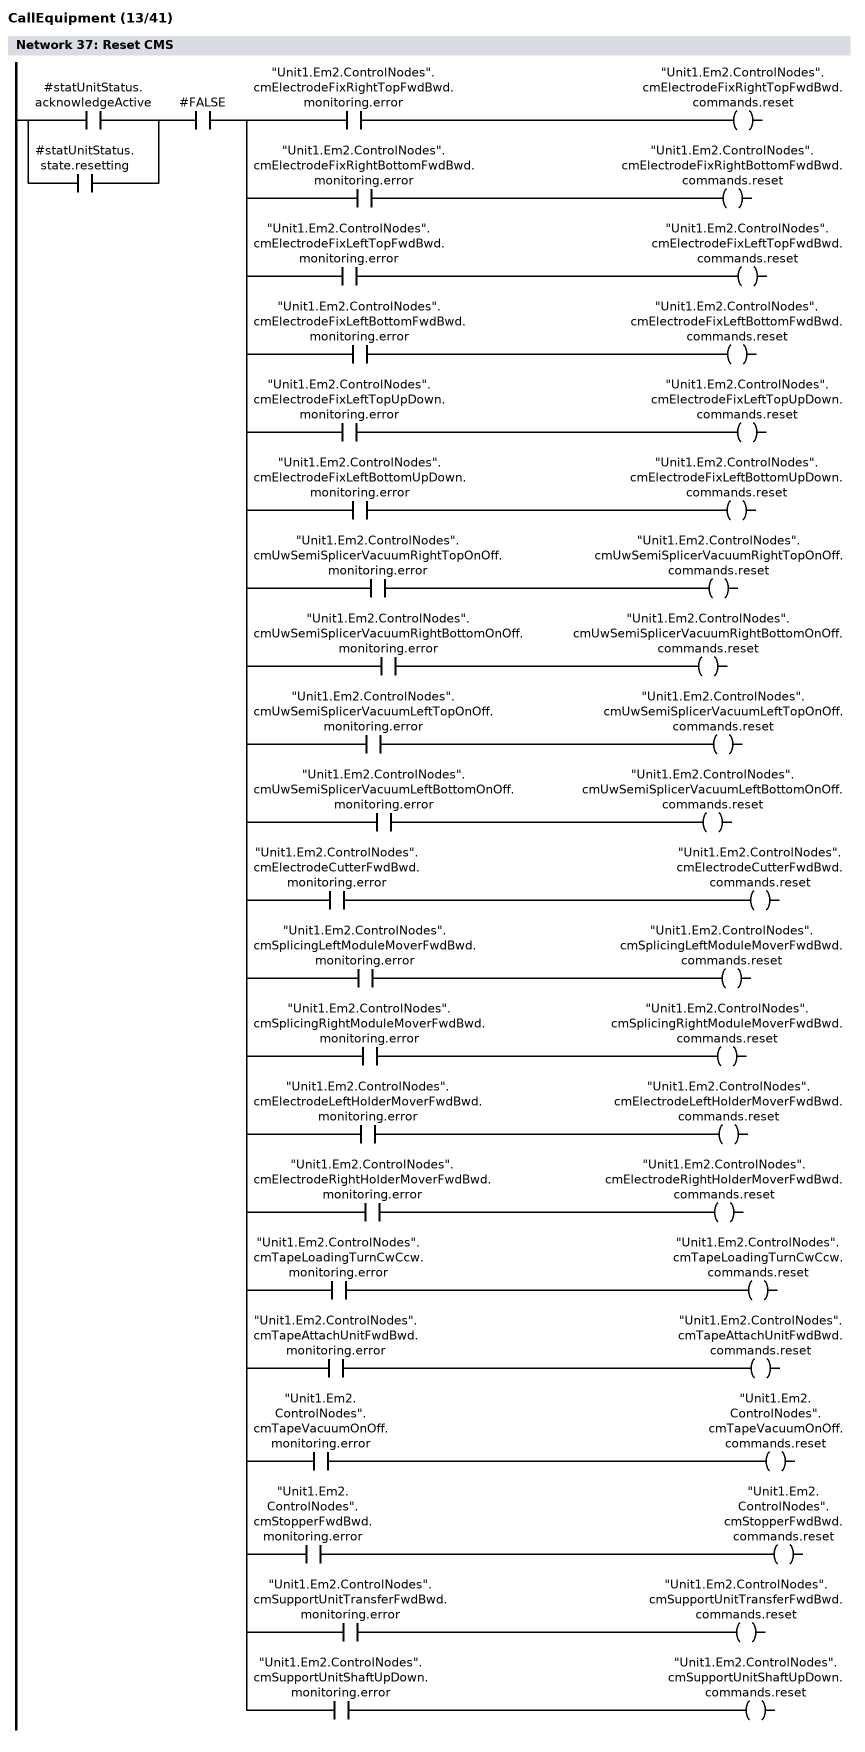
   RUNG wire#powerrail
      Contact( #statUnitStatus.acknowledgeActive )
      wire#w1
      Contact( #FALSE )
      wire#w2
      Contact( "Unit1.Em2.ControlNodes".cmElectrodeFixRightTopFwdBwd.monitoring.error )
      Coil( "Unit1.Em2.ControlNodes".cmElectrodeFixRightTopFwdBwd.commands.reset )
   END_RUNG
   RUNG wire#powerrail
      Contact( #statUnitStatus.state.resetting )
   END_RUNG wire#w1
   RUNG wire#w2
      Contact( "Unit1.Em2.ControlNodes".cmElectrodeFixRightBottomFwdBwd.monitoring.error )
      Coil( "Unit1.Em2.ControlNodes".cmElectrodeFixRightBottomFwdBwd.commands.reset )
   END_RUNG
   RUNG wire#w2
      Contact( "Unit1.Em2.ControlNodes".cmElectrodeFixLeftTopFwdBwd.monitoring.error )
      Coil( "Unit1.Em2.ControlNodes".cmElectrodeFixLeftTopFwdBwd.commands.reset )
   END_RUNG
   RUNG wire#w2
      Contact( "Unit1.Em2.ControlNodes".cmElectrodeFixLeftBottomFwdBwd.monitoring.error )
      Coil( "Unit1.Em2.ControlNodes".cmElectrodeFixLeftBottomFwdBwd.commands.reset )
   END_RUNG
   RUNG wire#w2
      Contact( "Unit1.Em2.ControlNodes".cmElectrodeFixLeftTopUpDown.monitoring.error )
      Coil( "Unit1.Em2.ControlNodes".cmElectrodeFixLeftTopUpDown.commands.reset )
   END_RUNG
   RUNG wire#w2
      Contact( "Unit1.Em2.ControlNodes".cmElectrodeFixLeftBottomUpDown.monitoring.error )
      Coil( "Unit1.Em2.ControlNodes".cmElectrodeFixLeftBottomUpDown.commands.reset )
   END_RUNG
   RUNG wire#w2
      Contact( "Unit1.Em2.ControlNodes".cmUwSemiSplicerVacuumRightTopOnOff.monitoring.error )
      Coil( "Unit1.Em2.ControlNodes".cmUwSemiSplicerVacuumRightTopOnOff.commands.reset )
   END_RUNG
   RUNG wire#w2
      Contact( "Unit1.Em2.ControlNodes".cmUwSemiSplicerVacuumRightBottomOnOff.monitoring.error )
      Coil( "Unit1.Em2.ControlNodes".cmUwSemiSplicerVacuumRightBottomOnOff.commands.reset )
   END_RUNG
   RUNG wire#w2
      Contact( "Unit1.Em2.ControlNodes".cmUwSemiSplicerVacuumLeftTopOnOff.monitoring.error )
      Coil( "Unit1.Em2.ControlNodes".cmUwSemiSplicerVacuumLeftTopOnOff.commands.reset )
   END_RUNG
   RUNG wire#w2
      Contact( "Unit1.Em2.ControlNodes".cmUwSemiSplicerVacuumLeftBottomOnOff.monitoring.error )
      Coil( "Unit1.Em2.ControlNodes".cmUwSemiSplicerVacuumLeftBottomOnOff.commands.reset )
   END_RUNG
   RUNG wire#w2
      Contact( "Unit1.Em2.ControlNodes".cmElectrodeCutterFwdBwd.monitoring.error )
      Coil( "Unit1.Em2.ControlNodes".cmElectrodeCutterFwdBwd.commands.reset )
   END_RUNG
   RUNG wire#w2
      Contact( "Unit1.Em2.ControlNodes".cmSplicingLeftModuleMoverFwdBwd.monitoring.error )
      Coil( "Unit1.Em2.ControlNodes".cmSplicingLeftModuleMoverFwdBwd.commands.reset )
   END_RUNG
   RUNG wire#w2
      Contact( "Unit1.Em2.ControlNodes".cmSplicingRightModuleMoverFwdBwd.monitoring.error )
      Coil( "Unit1.Em2.ControlNodes".cmSplicingRightModuleMoverFwdBwd.commands.reset )
   END_RUNG
   RUNG wire#w2
      Contact( "Unit1.Em2.ControlNodes".cmElectrodeLeftHolderMoverFwdBwd.monitoring.error )
      Coil( "Unit1.Em2.ControlNodes".cmElectrodeLeftHolderMoverFwdBwd.commands.reset )
   END_RUNG
   RUNG wire#w2
      Contact( "Unit1.Em2.ControlNodes".cmElectrodeRightHolderMoverFwdBwd.monitoring.error )
      Coil( "Unit1.Em2.ControlNodes".cmElectrodeRightHolderMoverFwdBwd.commands.reset )
   END_RUNG
   RUNG wire#w2
      Contact( "Unit1.Em2.ControlNodes".cmTapeLoadingTurnCwCcw.monitoring.error )
      Coil( "Unit1.Em2.ControlNodes".cmTapeLoadingTurnCwCcw.commands.reset )
   END_RUNG
   RUNG wire#w2
      Contact( "Unit1.Em2.ControlNodes".cmTapeAttachUnitFwdBwd.monitoring.error )
      Coil( "Unit1.Em2.ControlNodes".cmTapeAttachUnitFwdBwd.commands.reset )
   END_RUNG
   RUNG wire#w2
      Contact( "Unit1.Em2.ControlNodes".cmTapeVacuumOnOff.monitoring.error )
      Coil( "Unit1.Em2.ControlNodes".cmTapeVacuumOnOff.commands.reset )
   END_RUNG
   RUNG wire#w2
      Contact( "Unit1.Em2.ControlNodes".cmStopperFwdBwd.monitoring.error )
      Coil( "Unit1.Em2.ControlNodes".cmStopperFwdBwd.commands.reset )
   END_RUNG
   RUNG wire#w2
      Contact( "Unit1.Em2.ControlNodes".cmSupportUnitTransferFwdBwd.monitoring.error )
      Coil( "Unit1.Em2.ControlNodes".cmSupportUnitTransferFwdBwd.commands.reset )
   END_RUNG
   RUNG wire#w2
      Contact( "Unit1.Em2.ControlNodes".cmSupportUnitShaftUpDown.monitoring.error )
      Coil( "Unit1.Em2.ControlNodes".cmSupportUnitShaftUpDown.commands.reset )
   END_RUNG
   // the same network as SCL:
   #_w1 := (#statUnitStatus.acknowledgeActive OR #statUnitStatus.state.resetting) AND #FALSE;
   "Unit1.Em2.ControlNodes".cmElectrodeFixRightTopFwdBwd.commands.reset := #_w1 AND "Unit1.Em2.ControlNodes".cmElectrodeFixRightTopFwdBwd.monitoring.error;
   "Unit1.Em2.ControlNodes".cmElectrodeFixRightBottomFwdBwd.commands.reset := #_w1 AND "Unit1.Em2.ControlNodes".cmElectrodeFixRightBottomFwdBwd.monitoring.error;
   "Unit1.Em2.ControlNodes".cmElectrodeFixLeftTopFwdBwd.commands.reset := #_w1 AND "Unit1.Em2.ControlNodes".cmElectrodeFixLeftTopFwdBwd.monitoring.error;
   "Unit1.Em2.ControlNodes".cmElectrodeFixLeftBottomFwdBwd.commands.reset := #_w1 AND "Unit1.Em2.ControlNodes".cmElectrodeFixLeftBottomFwdBwd.monitoring.error;
   "Unit1.Em2.ControlNodes".cmElectrodeFixLeftTopUpDown.commands.reset := #_w1 AND "Unit1.Em2.ControlNodes".cmElectrodeFixLeftTopUpDown.monitoring.error;
   "Unit1.Em2.ControlNodes".cmElectrodeFixLeftBottomUpDown.commands.reset := #_w1 AND "Unit1.Em2.ControlNodes".cmElectrodeFixLeftBottomUpDown.monitoring.error;
   "Unit1.Em2.ControlNodes".cmUwSemiSplicerVacuumRightTopOnOff.commands.reset := #_w1 AND "Unit1.Em2.ControlNodes".cmUwSemiSplicerVacuumRightTopOnOff.monitoring.error;
   "Unit1.Em2.ControlNodes".cmUwSemiSplicerVacuumRightBottomOnOff.commands.reset := #_w1 AND "Unit1.Em2.ControlNodes".cmUwSemiSplicerVacuumRightBottomOnOff.monitoring.error;
   "Unit1.Em2.ControlNodes".cmUwSemiSplicerVacuumLeftTopOnOff.commands.reset := #_w1 AND "Unit1.Em2.ControlNodes".cmUwSemiSplicerVacuumLeftTopOnOff.monitoring.error;
   "Unit1.Em2.ControlNodes".cmUwSemiSplicerVacuumLeftBottomOnOff.commands.reset := #_w1 AND "Unit1.Em2.ControlNodes".cmUwSemiSplicerVacuumLeftBottomOnOff.monitoring.error;
   "Unit1.Em2.ControlNodes".cmElectrodeCutterFwdBwd.commands.reset := #_w1 AND "Unit1.Em2.ControlNodes".cmElectrodeCutterFwdBwd.monitoring.error;
   "Unit1.Em2.ControlNodes".cmSplicingLeftModuleMoverFwdBwd.commands.reset := #_w1 AND "Unit1.Em2.ControlNodes".cmSplicingLeftModuleMoverFwdBwd.monitoring.error;
   "Unit1.Em2.ControlNodes".cmSplicingRightModuleMoverFwdBwd.commands.reset := #_w1 AND "Unit1.Em2.ControlNodes".cmSplicingRightModuleMoverFwdBwd.monitoring.error;
   "Unit1.Em2.ControlNodes".cmElectrodeLeftHolderMoverFwdBwd.commands.reset := #_w1 AND "Unit1.Em2.ControlNodes".cmElectrodeLeftHolderMoverFwdBwd.monitoring.error;
   "Unit1.Em2.ControlNodes".cmElectrodeRightHolderMoverFwdBwd.commands.reset := #_w1 AND "Unit1.Em2.ControlNodes".cmElectrodeRightHolderMoverFwdBwd.monitoring.error;
   "Unit1.Em2.ControlNodes".cmTapeLoadingTurnCwCcw.commands.reset := #_w1 AND "Unit1.Em2.ControlNodes".cmTapeLoadingTurnCwCcw.monitoring.error;
   "Unit1.Em2.ControlNodes".cmTapeAttachUnitFwdBwd.commands.reset := #_w1 AND "Unit1.Em2.ControlNodes".cmTapeAttachUnitFwdBwd.monitoring.error;
   "Unit1.Em2.ControlNodes".cmTapeVacuumOnOff.commands.reset := #_w1 AND "Unit1.Em2.ControlNodes".cmTapeVacuumOnOff.monitoring.error;
   "Unit1.Em2.ControlNodes".cmStopperFwdBwd.commands.reset := #_w1 AND "Unit1.Em2.ControlNodes".cmStopperFwdBwd.monitoring.error;
   "Unit1.Em2.ControlNodes".cmSupportUnitTransferFwdBwd.commands.reset := #_w1 AND "Unit1.Em2.ControlNodes".cmSupportUnitTransferFwdBwd.monitoring.error;
   "Unit1.Em2.ControlNodes".cmSupportUnitShaftUpDown.commands.reset := #_w1 AND "Unit1.Em2.ControlNodes".cmSupportUnitShaftUpDown.monitoring.error;
END_REGION

REGION Network 38: CM Electrode Fix Right Top FWD/BWD Command Home
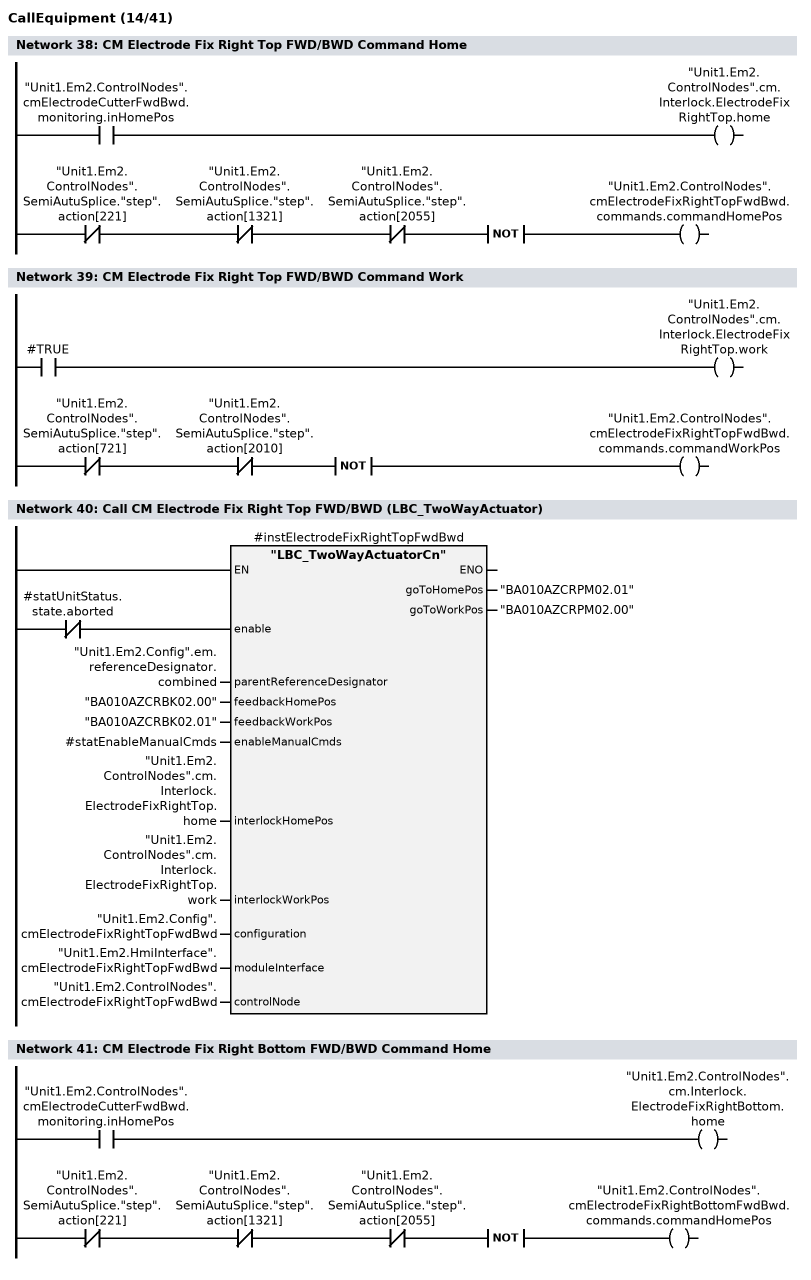
   RUNG wire#powerrail
      Contact( "Unit1.Em2.ControlNodes".cmElectrodeCutterFwdBwd.monitoring.inHomePos )
      Coil( "Unit1.Em2.ControlNodes".cm.Interlock.ElectrodeFixRightTop.home )
   END_RUNG
   RUNG wire#powerrail
      I_Contact( "Unit1.Em2.ControlNodes".SemiAutuSplice."step".action[221] )
      I_Contact( "Unit1.Em2.ControlNodes".SemiAutuSplice."step".action[1321] )
      I_Contact( "Unit1.Em2.ControlNodes".SemiAutuSplice."step".action[2055] )
      Not()
      Coil( "Unit1.Em2.ControlNodes".cmElectrodeFixRightTopFwdBwd.commands.commandHomePos )
   END_RUNG
   // the same network as SCL:
   "Unit1.Em2.ControlNodes".cm.Interlock.ElectrodeFixRightTop.home := "Unit1.Em2.ControlNodes".cmElectrodeCutterFwdBwd.monitoring.inHomePos;
   "Unit1.Em2.ControlNodes".cmElectrodeFixRightTopFwdBwd.commands.commandHomePos := NOT (NOT "Unit1.Em2.ControlNodes".SemiAutuSplice."step".action[221] AND NOT "Unit1.Em2.ControlNodes".SemiAutuSplice."step".action[1321] AND NOT "Unit1.Em2.ControlNodes".SemiAutuSplice."step".action[2055]);
END_REGION

REGION Network 39: CM Electrode Fix Right Top FWD/BWD Command Work
   RUNG wire#powerrail
      Contact( #TRUE )
      Coil( "Unit1.Em2.ControlNodes".cm.Interlock.ElectrodeFixRightTop.work )
   END_RUNG
   RUNG wire#powerrail
      I_Contact( "Unit1.Em2.ControlNodes".SemiAutuSplice."step".action[721] )
      I_Contact( "Unit1.Em2.ControlNodes".SemiAutuSplice."step".action[2010] )
      Not()
      Coil( "Unit1.Em2.ControlNodes".cmElectrodeFixRightTopFwdBwd.commands.commandWorkPos )
   END_RUNG
   // the same network as SCL:
   "Unit1.Em2.ControlNodes".cm.Interlock.ElectrodeFixRightTop.work := #TRUE;
   "Unit1.Em2.ControlNodes".cmElectrodeFixRightTopFwdBwd.commands.commandWorkPos := NOT (NOT "Unit1.Em2.ControlNodes".SemiAutuSplice."step".action[721] AND NOT "Unit1.Em2.ControlNodes".SemiAutuSplice."step".action[2010]);
END_REGION

REGION Network 40: Call CM Electrode Fix Right Top FWD/BWD (LBC_TwoWayActuator)
   RUNG wire#powerrail
      #instElectrodeFixRightTopFwdBwd(enable := wire#w1, parentReferenceDesignator := "Unit1.Em2.Config".em.referenceDesignator.combined, feedbackHomePos := "BA010AZCRBK02.00", feedbackWorkPos := "BA010AZCRBK02.01", enableManualCmds := #statEnableManualCmds, interlockHomePos := "Unit1.Em2.ControlNodes".cm.Interlock.ElectrodeFixRightTop.home, interlockWorkPos := "Unit1.Em2.ControlNodes".cm.Interlock.ElectrodeFixRightTop.work, configuration := "Unit1.Em2.Config".cmElectrodeFixRightTopFwdBwd, moduleInterface := "Unit1.Em2.HmiInterface".cmElectrodeFixRightTopFwdBwd, controlNode := "Unit1.Em2.ControlNodes".cmElectrodeFixRightTopFwdBwd, goToHomePos => "BA010AZCRPM02.01", goToWorkPos => "BA010AZCRPM02.00")
   END_RUNG
   RUNG wire#powerrail
      I_Contact( #statUnitStatus.state.aborted )
   END_RUNG wire#w1
   // the same network as SCL:
   #instElectrodeFixRightTopFwdBwd(enable := NOT #statUnitStatus.state.aborted,   // "LBC_TwoWayActuatorCn"
                           parentReferenceDesignator := "Unit1.Em2.Config".em.referenceDesignator.combined,
                           feedbackHomePos := "BA010AZCRBK02.00",
                           feedbackWorkPos := "BA010AZCRBK02.01",
                           enableManualCmds := #statEnableManualCmds,
                           interlockHomePos := "Unit1.Em2.ControlNodes".cm.Interlock.ElectrodeFixRightTop.home,
                           interlockWorkPos := "Unit1.Em2.ControlNodes".cm.Interlock.ElectrodeFixRightTop.work,
                           configuration := "Unit1.Em2.Config".cmElectrodeFixRightTopFwdBwd,
                           moduleInterface := "Unit1.Em2.HmiInterface".cmElectrodeFixRightTopFwdBwd,
                           controlNode := "Unit1.Em2.ControlNodes".cmElectrodeFixRightTopFwdBwd,
                           goToHomePos => "BA010AZCRPM02.01",
                           goToWorkPos => "BA010AZCRPM02.00");
END_REGION

REGION Network 41: CM Electrode Fix Right Bottom FWD/BWD Command Home
   RUNG wire#powerrail
      Contact( "Unit1.Em2.ControlNodes".cmElectrodeCutterFwdBwd.monitoring.inHomePos )
      Coil( "Unit1.Em2.ControlNodes".cm.Interlock.ElectrodeFixRightBottom.home )
   END_RUNG
   RUNG wire#powerrail
      I_Contact( "Unit1.Em2.ControlNodes".SemiAutuSplice."step".action[221] )
      I_Contact( "Unit1.Em2.ControlNodes".SemiAutuSplice."step".action[1321] )
      I_Contact( "Unit1.Em2.ControlNodes".SemiAutuSplice."step".action[2055] )
      Not()
      Coil( "Unit1.Em2.ControlNodes".cmElectrodeFixRightBottomFwdBwd.commands.commandHomePos )
   END_RUNG
   // the same network as SCL:
   "Unit1.Em2.ControlNodes".cm.Interlock.ElectrodeFixRightBottom.home := "Unit1.Em2.ControlNodes".cmElectrodeCutterFwdBwd.monitoring.inHomePos;
   "Unit1.Em2.ControlNodes".cmElectrodeFixRightBottomFwdBwd.commands.commandHomePos := NOT (NOT "Unit1.Em2.ControlNodes".SemiAutuSplice."step".action[221] AND NOT "Unit1.Em2.ControlNodes".SemiAutuSplice."step".action[1321] AND NOT "Unit1.Em2.ControlNodes".SemiAutuSplice."step".action[2055]);
END_REGION

REGION Network 42: CM Electrode Fix Right Bottom FWD/BWD Command Work
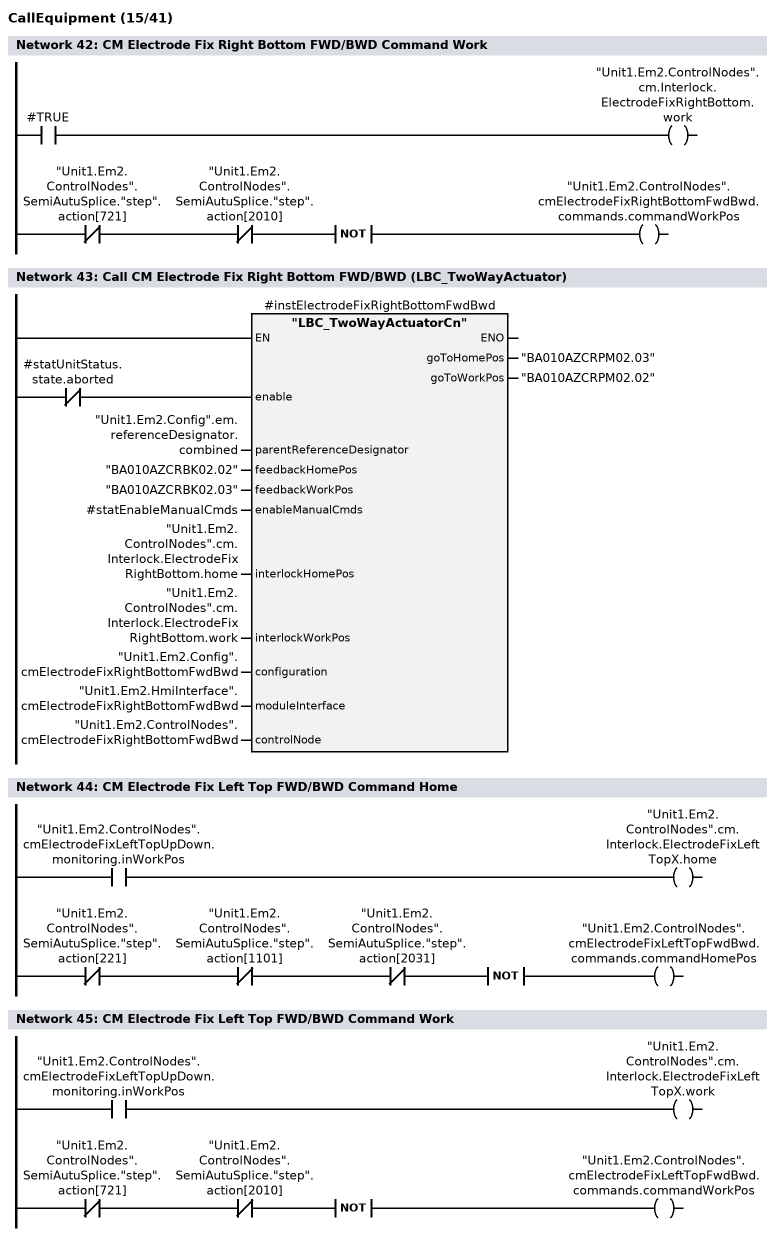
   RUNG wire#powerrail
      Contact( #TRUE )
      Coil( "Unit1.Em2.ControlNodes".cm.Interlock.ElectrodeFixRightBottom.work )
   END_RUNG
   RUNG wire#powerrail
      I_Contact( "Unit1.Em2.ControlNodes".SemiAutuSplice."step".action[721] )
      I_Contact( "Unit1.Em2.ControlNodes".SemiAutuSplice."step".action[2010] )
      Not()
      Coil( "Unit1.Em2.ControlNodes".cmElectrodeFixRightBottomFwdBwd.commands.commandWorkPos )
   END_RUNG
   // the same network as SCL:
   "Unit1.Em2.ControlNodes".cm.Interlock.ElectrodeFixRightBottom.work := #TRUE;
   "Unit1.Em2.ControlNodes".cmElectrodeFixRightBottomFwdBwd.commands.commandWorkPos := NOT (NOT "Unit1.Em2.ControlNodes".SemiAutuSplice."step".action[721] AND NOT "Unit1.Em2.ControlNodes".SemiAutuSplice."step".action[2010]);
END_REGION

REGION Network 43: Call CM Electrode Fix Right Bottom FWD/BWD (LBC_TwoWayActuator)
   RUNG wire#powerrail
      #instElectrodeFixRightBottomFwdBwd(enable := wire#w1, parentReferenceDesignator := "Unit1.Em2.Config".em.referenceDesignator.combined, feedbackHomePos := "BA010AZCRBK02.02", feedbackWorkPos := "BA010AZCRBK02.03", enableManualCmds := #statEnableManualCmds, interlockHomePos := "Unit1.Em2.ControlNodes".cm.Interlock.ElectrodeFixRightBottom.home, interlockWorkPos := "Unit1.Em2.ControlNodes".cm.Interlock.ElectrodeFixRightBottom.work, configuration := "Unit1.Em2.Config".cmElectrodeFixRightBottomFwdBwd, moduleInterface := "Unit1.Em2.HmiInterface".cmElectrodeFixRightBottomFwdBwd, controlNode := "Unit1.Em2.ControlNodes".cmElectrodeFixRightBottomFwdBwd, goToHomePos => "BA010AZCRPM02.03", goToWorkPos => "BA010AZCRPM02.02")
   END_RUNG
   RUNG wire#powerrail
      I_Contact( #statUnitStatus.state.aborted )
   END_RUNG wire#w1
   // the same network as SCL:
   #instElectrodeFixRightBottomFwdBwd(enable := NOT #statUnitStatus.state.aborted,   // "LBC_TwoWayActuatorCn"
                           parentReferenceDesignator := "Unit1.Em2.Config".em.referenceDesignator.combined,
                           feedbackHomePos := "BA010AZCRBK02.02",
                           feedbackWorkPos := "BA010AZCRBK02.03",
                           enableManualCmds := #statEnableManualCmds,
                           interlockHomePos := "Unit1.Em2.ControlNodes".cm.Interlock.ElectrodeFixRightBottom.home,
                           interlockWorkPos := "Unit1.Em2.ControlNodes".cm.Interlock.ElectrodeFixRightBottom.work,
                           configuration := "Unit1.Em2.Config".cmElectrodeFixRightBottomFwdBwd,
                           moduleInterface := "Unit1.Em2.HmiInterface".cmElectrodeFixRightBottomFwdBwd,
                           controlNode := "Unit1.Em2.ControlNodes".cmElectrodeFixRightBottomFwdBwd,
                           goToHomePos => "BA010AZCRPM02.03",
                           goToWorkPos => "BA010AZCRPM02.02");
END_REGION

REGION Network 44: CM Electrode Fix Left Top FWD/BWD Command Home
   RUNG wire#powerrail
      Contact( "Unit1.Em2.ControlNodes".cmElectrodeFixLeftTopUpDown.monitoring.inWorkPos )
      Coil( "Unit1.Em2.ControlNodes".cm.Interlock.ElectrodeFixLeftTopX.home )
   END_RUNG
   RUNG wire#powerrail
      I_Contact( "Unit1.Em2.ControlNodes".SemiAutuSplice."step".action[221] )
      I_Contact( "Unit1.Em2.ControlNodes".SemiAutuSplice."step".action[1101] )
      I_Contact( "Unit1.Em2.ControlNodes".SemiAutuSplice."step".action[2031] )
      Not()
      Coil( "Unit1.Em2.ControlNodes".cmElectrodeFixLeftTopFwdBwd.commands.commandHomePos )
   END_RUNG
   // the same network as SCL:
   "Unit1.Em2.ControlNodes".cm.Interlock.ElectrodeFixLeftTopX.home := "Unit1.Em2.ControlNodes".cmElectrodeFixLeftTopUpDown.monitoring.inWorkPos;
   "Unit1.Em2.ControlNodes".cmElectrodeFixLeftTopFwdBwd.commands.commandHomePos := NOT (NOT "Unit1.Em2.ControlNodes".SemiAutuSplice."step".action[221] AND NOT "Unit1.Em2.ControlNodes".SemiAutuSplice."step".action[1101] AND NOT "Unit1.Em2.ControlNodes".SemiAutuSplice."step".action[2031]);
END_REGION

REGION Network 45: CM Electrode Fix Left Top FWD/BWD Command Work
   RUNG wire#powerrail
      Contact( "Unit1.Em2.ControlNodes".cmElectrodeFixLeftTopUpDown.monitoring.inWorkPos )
      Coil( "Unit1.Em2.ControlNodes".cm.Interlock.ElectrodeFixLeftTopX.work )
   END_RUNG
   RUNG wire#powerrail
      I_Contact( "Unit1.Em2.ControlNodes".SemiAutuSplice."step".action[721] )
      I_Contact( "Unit1.Em2.ControlNodes".SemiAutuSplice."step".action[2010] )
      Not()
      Coil( "Unit1.Em2.ControlNodes".cmElectrodeFixLeftTopFwdBwd.commands.commandWorkPos )
   END_RUNG
   // the same network as SCL:
   "Unit1.Em2.ControlNodes".cm.Interlock.ElectrodeFixLeftTopX.work := "Unit1.Em2.ControlNodes".cmElectrodeFixLeftTopUpDown.monitoring.inWorkPos;
   "Unit1.Em2.ControlNodes".cmElectrodeFixLeftTopFwdBwd.commands.commandWorkPos := NOT (NOT "Unit1.Em2.ControlNodes".SemiAutuSplice."step".action[721] AND NOT "Unit1.Em2.ControlNodes".SemiAutuSplice."step".action[2010]);
END_REGION

REGION Network 46: Call CM Electrode Fix Left Top FWD/BWD (LBC_TwoWayActuator)
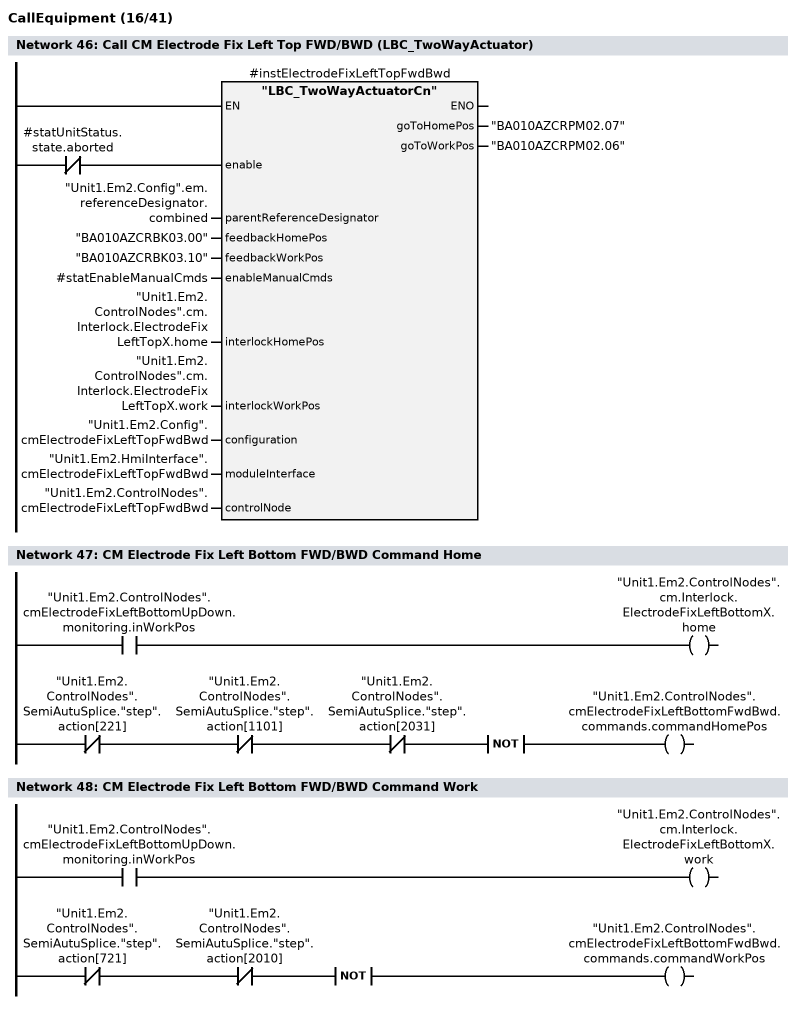
   RUNG wire#powerrail
      #instElectrodeFixLeftTopFwdBwd(enable := wire#w1, parentReferenceDesignator := "Unit1.Em2.Config".em.referenceDesignator.combined, feedbackHomePos := "BA010AZCRBK03.00", feedbackWorkPos := "BA010AZCRBK03.10", enableManualCmds := #statEnableManualCmds, interlockHomePos := "Unit1.Em2.ControlNodes".cm.Interlock.ElectrodeFixLeftTopX.home, interlockWorkPos := "Unit1.Em2.ControlNodes".cm.Interlock.ElectrodeFixLeftTopX.work, configuration := "Unit1.Em2.Config".cmElectrodeFixLeftTopFwdBwd, moduleInterface := "Unit1.Em2.HmiInterface".cmElectrodeFixLeftTopFwdBwd, controlNode := "Unit1.Em2.ControlNodes".cmElectrodeFixLeftTopFwdBwd, goToHomePos => "BA010AZCRPM02.07", goToWorkPos => "BA010AZCRPM02.06")
   END_RUNG
   RUNG wire#powerrail
      I_Contact( #statUnitStatus.state.aborted )
   END_RUNG wire#w1
   // the same network as SCL:
   #instElectrodeFixLeftTopFwdBwd(enable := NOT #statUnitStatus.state.aborted,   // "LBC_TwoWayActuatorCn"
                           parentReferenceDesignator := "Unit1.Em2.Config".em.referenceDesignator.combined,
                           feedbackHomePos := "BA010AZCRBK03.00",
                           feedbackWorkPos := "BA010AZCRBK03.10",
                           enableManualCmds := #statEnableManualCmds,
                           interlockHomePos := "Unit1.Em2.ControlNodes".cm.Interlock.ElectrodeFixLeftTopX.home,
                           interlockWorkPos := "Unit1.Em2.ControlNodes".cm.Interlock.ElectrodeFixLeftTopX.work,
                           configuration := "Unit1.Em2.Config".cmElectrodeFixLeftTopFwdBwd,
                           moduleInterface := "Unit1.Em2.HmiInterface".cmElectrodeFixLeftTopFwdBwd,
                           controlNode := "Unit1.Em2.ControlNodes".cmElectrodeFixLeftTopFwdBwd,
                           goToHomePos => "BA010AZCRPM02.07",
                           goToWorkPos => "BA010AZCRPM02.06");
END_REGION

REGION Network 47: CM Electrode Fix Left Bottom FWD/BWD Command Home
   RUNG wire#powerrail
      Contact( "Unit1.Em2.ControlNodes".cmElectrodeFixLeftBottomUpDown.monitoring.inWorkPos )
      Coil( "Unit1.Em2.ControlNodes".cm.Interlock.ElectrodeFixLeftBottomX.home )
   END_RUNG
   RUNG wire#powerrail
      I_Contact( "Unit1.Em2.ControlNodes".SemiAutuSplice."step".action[221] )
      I_Contact( "Unit1.Em2.ControlNodes".SemiAutuSplice."step".action[1101] )
      I_Contact( "Unit1.Em2.ControlNodes".SemiAutuSplice."step".action[2031] )
      Not()
      Coil( "Unit1.Em2.ControlNodes".cmElectrodeFixLeftBottomFwdBwd.commands.commandHomePos )
   END_RUNG
   // the same network as SCL:
   "Unit1.Em2.ControlNodes".cm.Interlock.ElectrodeFixLeftBottomX.home := "Unit1.Em2.ControlNodes".cmElectrodeFixLeftBottomUpDown.monitoring.inWorkPos;
   "Unit1.Em2.ControlNodes".cmElectrodeFixLeftBottomFwdBwd.commands.commandHomePos := NOT (NOT "Unit1.Em2.ControlNodes".SemiAutuSplice."step".action[221] AND NOT "Unit1.Em2.ControlNodes".SemiAutuSplice."step".action[1101] AND NOT "Unit1.Em2.ControlNodes".SemiAutuSplice."step".action[2031]);
END_REGION

REGION Network 48: CM Electrode Fix Left Bottom FWD/BWD Command Work
   RUNG wire#powerrail
      Contact( "Unit1.Em2.ControlNodes".cmElectrodeFixLeftBottomUpDown.monitoring.inWorkPos )
      Coil( "Unit1.Em2.ControlNodes".cm.Interlock.ElectrodeFixLeftBottomX.work )
   END_RUNG
   RUNG wire#powerrail
      I_Contact( "Unit1.Em2.ControlNodes".SemiAutuSplice."step".action[721] )
      I_Contact( "Unit1.Em2.ControlNodes".SemiAutuSplice."step".action[2010] )
      Not()
      Coil( "Unit1.Em2.ControlNodes".cmElectrodeFixLeftBottomFwdBwd.commands.commandWorkPos )
   END_RUNG
   // the same network as SCL:
   "Unit1.Em2.ControlNodes".cm.Interlock.ElectrodeFixLeftBottomX.work := "Unit1.Em2.ControlNodes".cmElectrodeFixLeftBottomUpDown.monitoring.inWorkPos;
   "Unit1.Em2.ControlNodes".cmElectrodeFixLeftBottomFwdBwd.commands.commandWorkPos := NOT (NOT "Unit1.Em2.ControlNodes".SemiAutuSplice."step".action[721] AND NOT "Unit1.Em2.ControlNodes".SemiAutuSplice."step".action[2010]);
END_REGION

REGION Network 49: Call CM Electrode Fix Left Bottom FWD/BWD (LBC_TwoWayActuator)
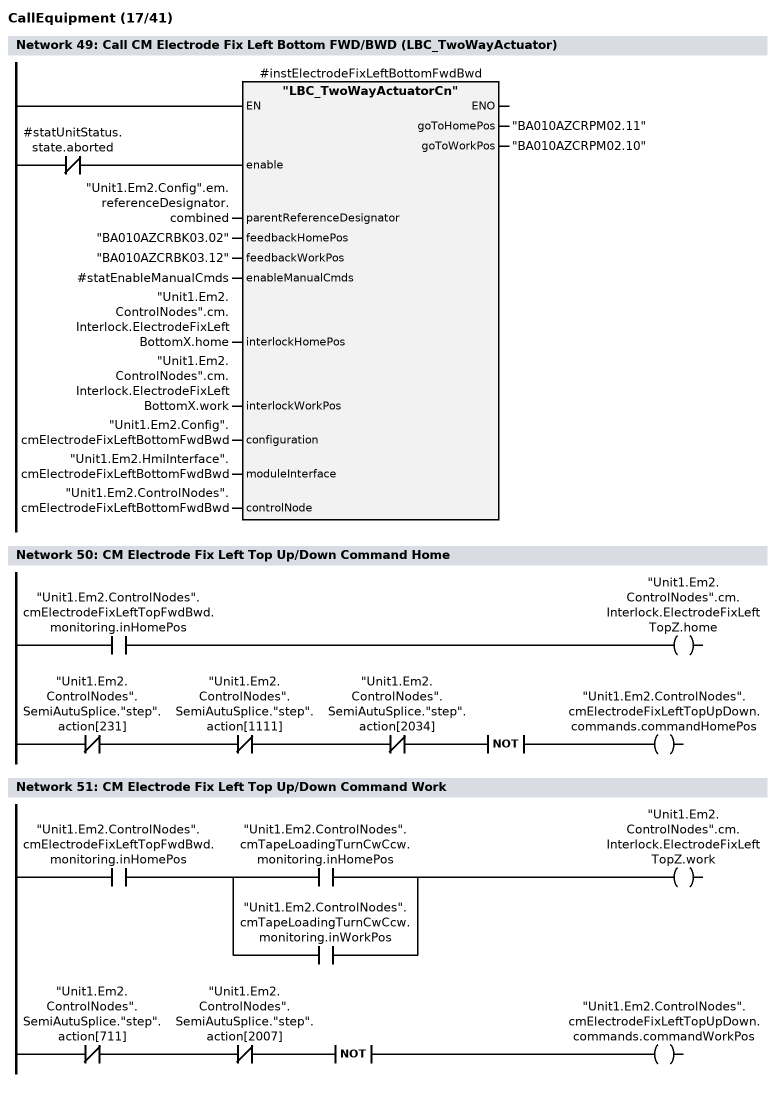
   RUNG wire#powerrail
      #instElectrodeFixLeftBottomFwdBwd(enable := wire#w1, parentReferenceDesignator := "Unit1.Em2.Config".em.referenceDesignator.combined, feedbackHomePos := "BA010AZCRBK03.02", feedbackWorkPos := "BA010AZCRBK03.12", enableManualCmds := #statEnableManualCmds, interlockHomePos := "Unit1.Em2.ControlNodes".cm.Interlock.ElectrodeFixLeftBottomX.home, interlockWorkPos := "Unit1.Em2.ControlNodes".cm.Interlock.ElectrodeFixLeftBottomX.work, configuration := "Unit1.Em2.Config".cmElectrodeFixLeftBottomFwdBwd, moduleInterface := "Unit1.Em2.HmiInterface".cmElectrodeFixLeftBottomFwdBwd, controlNode := "Unit1.Em2.ControlNodes".cmElectrodeFixLeftBottomFwdBwd, goToHomePos => "BA010AZCRPM02.11", goToWorkPos => "BA010AZCRPM02.10")
   END_RUNG
   RUNG wire#powerrail
      I_Contact( #statUnitStatus.state.aborted )
   END_RUNG wire#w1
   // the same network as SCL:
   #instElectrodeFixLeftBottomFwdBwd(enable := NOT #statUnitStatus.state.aborted,   // "LBC_TwoWayActuatorCn"
                           parentReferenceDesignator := "Unit1.Em2.Config".em.referenceDesignator.combined,
                           feedbackHomePos := "BA010AZCRBK03.02",
                           feedbackWorkPos := "BA010AZCRBK03.12",
                           enableManualCmds := #statEnableManualCmds,
                           interlockHomePos := "Unit1.Em2.ControlNodes".cm.Interlock.ElectrodeFixLeftBottomX.home,
                           interlockWorkPos := "Unit1.Em2.ControlNodes".cm.Interlock.ElectrodeFixLeftBottomX.work,
                           configuration := "Unit1.Em2.Config".cmElectrodeFixLeftBottomFwdBwd,
                           moduleInterface := "Unit1.Em2.HmiInterface".cmElectrodeFixLeftBottomFwdBwd,
                           controlNode := "Unit1.Em2.ControlNodes".cmElectrodeFixLeftBottomFwdBwd,
                           goToHomePos => "BA010AZCRPM02.11",
                           goToWorkPos => "BA010AZCRPM02.10");
END_REGION

REGION Network 50: CM Electrode Fix Left Top Up/Down Command Home
   RUNG wire#powerrail
      Contact( "Unit1.Em2.ControlNodes".cmElectrodeFixLeftTopFwdBwd.monitoring.inHomePos )
      Coil( "Unit1.Em2.ControlNodes".cm.Interlock.ElectrodeFixLeftTopZ.home )
   END_RUNG
   RUNG wire#powerrail
      I_Contact( "Unit1.Em2.ControlNodes".SemiAutuSplice."step".action[231] )
      I_Contact( "Unit1.Em2.ControlNodes".SemiAutuSplice."step".action[1111] )
      I_Contact( "Unit1.Em2.ControlNodes".SemiAutuSplice."step".action[2034] )
      Not()
      Coil( "Unit1.Em2.ControlNodes".cmElectrodeFixLeftTopUpDown.commands.commandHomePos )
   END_RUNG
   // the same network as SCL:
   "Unit1.Em2.ControlNodes".cm.Interlock.ElectrodeFixLeftTopZ.home := "Unit1.Em2.ControlNodes".cmElectrodeFixLeftTopFwdBwd.monitoring.inHomePos;
   "Unit1.Em2.ControlNodes".cmElectrodeFixLeftTopUpDown.commands.commandHomePos := NOT (NOT "Unit1.Em2.ControlNodes".SemiAutuSplice."step".action[231] AND NOT "Unit1.Em2.ControlNodes".SemiAutuSplice."step".action[1111] AND NOT "Unit1.Em2.ControlNodes".SemiAutuSplice."step".action[2034]);
END_REGION

REGION Network 51: CM Electrode Fix Left Top Up/Down Command Work
   RUNG wire#powerrail
      Contact( "Unit1.Em2.ControlNodes".cmElectrodeFixLeftTopFwdBwd.monitoring.inHomePos )
      wire#w1
      Contact( "Unit1.Em2.ControlNodes".cmTapeLoadingTurnCwCcw.monitoring.inHomePos )
      wire#w2
      Coil( "Unit1.Em2.ControlNodes".cm.Interlock.ElectrodeFixLeftTopZ.work )
   END_RUNG
   RUNG wire#w1
      Contact( "Unit1.Em2.ControlNodes".cmTapeLoadingTurnCwCcw.monitoring.inWorkPos )
   END_RUNG wire#w2
   RUNG wire#powerrail
      I_Contact( "Unit1.Em2.ControlNodes".SemiAutuSplice."step".action[711] )
      I_Contact( "Unit1.Em2.ControlNodes".SemiAutuSplice."step".action[2007] )
      Not()
      Coil( "Unit1.Em2.ControlNodes".cmElectrodeFixLeftTopUpDown.commands.commandWorkPos )
   END_RUNG
   // the same network as SCL:
   "Unit1.Em2.ControlNodes".cm.Interlock.ElectrodeFixLeftTopZ.work := "Unit1.Em2.ControlNodes".cmElectrodeFixLeftTopFwdBwd.monitoring.inHomePos AND ("Unit1.Em2.ControlNodes".cmTapeLoadingTurnCwCcw.monitoring.inHomePos OR "Unit1.Em2.ControlNodes".cmTapeLoadingTurnCwCcw.monitoring.inWorkPos);
   "Unit1.Em2.ControlNodes".cmElectrodeFixLeftTopUpDown.commands.commandWorkPos := NOT (NOT "Unit1.Em2.ControlNodes".SemiAutuSplice."step".action[711] AND NOT "Unit1.Em2.ControlNodes".SemiAutuSplice."step".action[2007]);
END_REGION

